	Ca_Quantited:UINT;//负极已叠数量
	Ca_KDQuantited:UINT;//负极空叠隔膜已叠片数
	Ca_EmptyRunKDQuantited:UINT;//负极空跑模式空叠隔膜已叠层数
	Ca_CarryingFalg:BOOL;//负极搬运吸盘有无料标记
	Ca_SegbeltFalg:BOOL;//负极段皮带取模切机械手有无料标记
	Ca_deviationFalg:BOOL;//负极纠偏平台有无料标记
	Ca_DPCarryingFalg:BOOL;//负极叠台搬运吸盘有无料标记
	Ca_DPRequest:BOOL;//负极叠片请求
	//Ca_deviationCCDOK:BOOL;//负极纠偏平台拍照OK
	//Ca_deviationCCDNG:BOOL;//负极纠偏平台拍照NG	
	Ca_deviationCCDDone:BOOL;//负极纠偏平台拍照完成
	Ca_CCDStart:BOOL;//CCD拍照启动
	//Ca_BlueflagingKDSet:UINT;//负极接带空叠隔膜设定片数
	//Ca_YellowmarkKDSet:UINT;//负极色标空叠隔膜设定片数
	Ca_Blueflaging_TF:UINT;//负极蓝胶标记空叠层数		

	Ca_deviationFPOK:BOOL;//负极纠偏平台允许放极片
	Ca_deviationDPOK:BOOL;//负极纠偏平台允许取极片
	Ca_deviationDone:BOOL;//负极纠偏平台纠偏完成
	Ca_CacheBeltDLOK:BOOL;//负极流水线缓存皮带允许取极片
	Ca_CacheBelting:BOOL;//负极流水线缓存皮带取极片中
	Ca_CacheBeltFLOK:BOOL;//负极流水线缓存皮带允许放极片
	Ca_CacheBeltFLing:BOOL;//负极流水线缓存皮带放极片中
	Ca_MainBeltOK:BOOL;//负极流水线主分料皮带允许取极片
	Ca_MainBelting:BOOL;//负极流水线主分料皮带取极片中
	Ca_betlMoveOK:BOOL;//负极搬运升降1在安全位、负极搬运升降2在安全位允许负极流水线线皮带移动
	Ca_AxisCarrying:BOOL;//负极各轴正在运行到初始位中	
	Ca_BeltDone:BOOL;//正极取主分料流水线极片完成
	Ca_BeltSafe:BOOL;//正极取主分料流水线极片安全位
	GetPiceReady:BOOL;//负  极 准备好取分段流水线上的极片
	JumpPiceReady:BOOL;//负  极 放弃取分段流水线上的极片
	bCa_PoleHave:BOOL;//负极取料位无片
	
	Ca_StandbyStep:ARRAY[0..9] OF UINT;//负极备极片程序步
	CarryingSafepos:ARRAY[0..9] OF BOOL;//负极搬动轴在安全位置指示
	Error:ARRAY[0..80] OF BOOL;//报警
		Error_tips	:ARRAY[0..60] OF BOOL;//报警提示
	
	RectifydevStart:BOOL; //纠偏启动
	RectifydevDone:BOOL; //纠偏完成
	//CCD_X1:REAL; //纠偏平台X1的纠偏量
	//CCD_X2:REAL;//纠偏平台X2的纠偏量
	//CCD_Y:REAL;//纠偏平台Y的纠偏量	
	
	DemarcateStart:BOOL; //标定启动	
	DemarcateDone:BOOL; //CCD标定完成
	Demarcateing:BOOL;//CCD标定中
	
	CreateCamStart:BOOL;//负极取片凸轮创建启动
	CreateCamDone:BOOL;//负极取片凸轮创建完成
	
	bCaCCD_TestDo:BOOL;//负极CCD测试开始
	iCaCCD_PhotoCT:INT;//负极拍照取图时间
	iCaCCD_RectifyCT:INT;//负极纠偏时间	
	Ca_CCD_amount :INT;//负极连续NG计数
	Ca_DTqr :BOOL;//负极极片掉片人工确认按钮
	Ca_Rectifydev_CQ :BOOL;//负极纠偏平台除尘
	Ca_Rectifydev_CS :INT;//纠偏计数
	
	Ca_Rectifydev_PB :BOOL;//二次纠偏屏蔽 OFF:屏蔽二次纠偏
	Ca_VacuumErrorNG :BOOL;//负极抛真空NG料标志
	//新增，首层隔膜
	Ca_FirstFoldCnt:INT;//负极首层隔膜已叠次数
	Ca_FirstFoldSet:INT:=1;//负极首层隔膜设定次数
	//20240414WCZ
	RectifyTryStart:BOOL;//CCD重复精度测试启动
	SuckerTestStart:BOOL;//吸盘重复精度测试启动
END_STRUCT
END_TYPE

// ---- P2DUTs/39User2/conDT_Date.TcDUT
TYPE conDT_Date ://叠台叠片
STRUCT
	
	bRecDevBtn:BOOL;//隔膜检测传感器标定按钮
	DT_Blue_TF		  :BOOL;//蓝胶踢废		OFF:屏蔽
	Yellowmark_TF:BOOL;//隔膜色标踢废
	DTIniti_Hbtn:BOOL;//叠台初始化，触摸屏按钮
	DTIniti_Done:BOOL;//叠台初始化完成
	DT_AutoHMI:BOOL;//叠台触摸屏自动
	DT_ManuaHMI:BOOL;//叠台触摸屏手动	
	
	ALLIniti_Hbtn:BOOL;//叠片回原点启动，触摸屏按M钮
	ALLIniti_Done:BOOL;//叠片回原点完成
	CWW:BOOL; //纠偏方向选择
	RecDevEqupos:REAL; //纠偏传感器平衡位置
	RecDevPV:REAL;//纠偏传感器当前值
	RecDevPV1:REAL;//纠偏传感器当前值
	Error:ARRAY[0..100] OF BOOL;//报警
	DT_camError:BOOL;//叠台凸轮报警需初始化
	
	BluGlueNG:ARRAY[0..1] OF BOOL;//表示蓝胶当前电芯或下个电芯NG
	
	CreateCamStart1:BOOL;//叠台压刀凸轮创建启动
	CreateCamDone1:BOOL;//叠台压刀凸轮创建完成
	CreateCamStart2:BOOL;//叠台缓存凸轮创建启动
	CreateCamDone2:BOOL;//叠台缓存凸轮创建完成
	
	Step:ARRAY[0..9] OF UINT;//程序步
	SinStepMode:BOOL;//单步模式
	DP_Mode:BOOL;//叠片完成后，空叠隔膜
	DT_Chesoe:BOOL;//叠负极片选择 
	DT_CellNG_TF	  :BOOL;//对齐度NG梯度踢废 OFF:屏蔽
	
	
	OffloadRequest:BOOL;//叠电芯完成请求下货
	OffloadDone:BOOL;//叠台下货完成
	
	rTension_Start:BOOL;//一键张力启动
	bTenExecute:BOOL;//隔膜张力启动
	bStudyExecute:BOOL;//隔膜张力学习
	PidSwitch:BOOL:=TRUE;//被动放卷开关选择
	fWindDiameter:REAL;//隔膜放卷轴当前卷径
	bTenReady:BOOL;//张力准备好
	bTensionOK:BOOL;//张力OK
	bTenCcw:BOOL;//放卷方向选择
	PTenidSwitch:BOOL;//张力PID开关
	TenAnglePos:REAL;//张力摆杆当前角度	
	TeniGMMoveCount:DINT;//隔膜同步拉伸次数
	
	RectifydevStarte:BOOL;//隔膜纠偏开启HMI
	RectifydevModel:BOOL;//隔膜纠偏屏蔽
	ClearCount:BOOL;//正、负极清零
	
	CDD_OverStart:BOOL;//CCD对奇度检测
	CDD_OverStart_First:BOOL;//CCD对奇度检测压刀间距测量拍照
	OverhandResult:INT;//叠台极片检测有无
	OverhandFirstPice:INT;//叠台极片首层标记
	iOverError:INT;//对齐度检测报警	1：OK，2：NG    实时检测，检测到结果为2就报警

	
	DT_Start           :BOOL;//叠台启动
	
	DT_coumtHight:REAL;//叠片叠台升降已下降高度
	DT_CCD_TwoModel:BOOL;//叠台CCD拍照复检模式
	Door_error :ARRAY[0..80] OF BOOL;//叠台门禁报警
	DT_AllCamOut:BOOL;//叠台一键解耦
	DT_Memory   :INT;//叠台电芯记忆
	DT_amount   :UINT;//已叠电芯数
	DT_amount_clear :BOOL;//电芯数清零
	DT_No      :STRING;//叠台编号
	Machine_No: STRING;//机台编号
	//Cell_Hough    :INT;//(CCD综合评定结果/对齐度)1、对齐度OK，2、对齐度NG
	fWindDiameter_min :REAL;//最小卷径
	Door_Forbidden   :BOOL;//门禁禁用
	Dust_name :INT;//送片皮带毛刷电机
	DiaphragmUnwindingTension :REAL;//隔膜张力
	Manual	:BOOL;//叠台手动
	Put_time :STRING;//投入时间
	DT_Overhang : BOOL;//对齐度屏蔽
	CCD_Overhang_button :BOOL;//叠台电芯确认无极片按钮
	DT_Oerhang_Z :INT;//对齐度结果
	Overhang_TF :BOOL;//对齐度NG踢废信号
	Overhang_Warm:BOOL;//对齐度超限报警
	Overhang_Warm_Reset:BOOL;
	DT_QLqr :BOOL;//叠台已叠片数清零弹窗
	DT_init_OK :BOOL;//叠台工位初始位完成
	YD_JS_L_clear :BOOL;//左压刀计数清零
	YD_JS_R_clear :BOOL;//右压刀计数清零	
	stBnt_Blueflag:BOOL;//蓝胶标记启动
	BlueflagBnt_Warm:BOOL;//是否启动蓝胶标记提示
	
	DT_DayHough:REAL;//对齐度NG数统计白班
	DT_DayHoughAn:REAL;//白班对齐度NG踢废正极片数
	DT_DayHoughCa:REAL;//白班对齐度NG踢废负极片数
	DT_NightHough:REAL;//对齐度NG数统计晚班
	DT_NightHoughAn:REAL;//夜班对齐度NG踢废正极片数
	DT_NightHoughCa:REAL;//夜班对齐度NG踢废负极片数
	DT_DayHough_U:UINT;//对齐度NG数统计白班整数
	DT_NightHough_U:UINT;//对齐度NG数统计晚班整数
	
	DTJD_DayHough:REAL;//白班接带对齐度NG数统计
	DTJD_DayHoughAn:REAL;//白班接带对齐度NG踢废正极片数
	DTJD_DayHoughCa:REAL;//白班接带对齐度NG踢废负极片数
	DTJD_NightHough:REAL;//夜班接带对齐度NG数统计
	DTJD_NightHoughAn:REAL;//夜班接带对齐度NG踢废正极片数
	DTJD_NightHoughCa:REAL;//夜班接带对齐度NG踢废负极片数
	DTJD_DayHough_U:UINT;//白班接带对齐度NG数统计整数
	DTJD_NightHough_U:UINT;//夜班接带对齐度NG数统计整数
	
	DT_GMchange:BOOL;//隔膜更换时间
	DT_OverhangNG:BOOL;//对齐度NG下料时间
	Query:BOOL;//时间查询
	date1:INT;//查询日期
	
	//20231216新增叠台各种状态
	iDTRunStatus:INT;//叠台运行状态：1:自动	2：手动	3：正常电芯空叠隔膜中	4:下料	5：空跑(空叠隔膜)	6:正极踢废		7：负极踢废
	FirstEmpFold:BOOL;//首层空叠隔膜屏蔽

	//20240102新增
	HMI_WinBtn:ARRAY[1..50] OF BOOL;//触摸屏弹窗确认按钮
	HMI_WinOEE_Btn:ARRAY[1..50] OF BOOL;//OEE采集确认按钮
	DiaphragmPartNumberOK    :BOOL;   //隔膜料号OK
	BluePartNumberOK    :BOOL;   //蓝胶料号OK
	PartNumberOff       :BOOL;   //料号功能屏蔽
	Error_tips	:ARRAY[1..30] OF BOOL;//报警提示
	
	fWindLength_M:REAL; //隔膜放卷轴当前米数
	DT_DebugMode           :BOOL;//叠台调试模式料
	DT_Sheetkick     :BOOL;//对齐度单片踢废屏蔽
	DT_YDOpenwindow  :BOOL;//叠台压刀开窗测量屏蔽
	DT_OHclosure		:BOOL;		//对齐度闭环屏蔽		ON是屏蔽
	GMAngleALMsel     :BOOL;		//隔膜卷径报警屏蔽		ON是屏蔽
	
	YD_ferrJSclear :BOOL;//压刀铁氟龙计数清零
	An_sucker1_JSclear      :BOOL;//正极送片搬运吸盘计数清零  
    An_sucker2_JSclear      :BOOL;//正极叠台搬运吸盘计数清零  
    Ca_sucker1_JSclear      :BOOL;//负极送片搬运吸盘计数清零  
    Ca_sucker2_JSclear      :BOOL;//负极叠台搬运吸盘计数清零  
    Ca_sucker3_JSclear      :BOOL;//负极流水线搬运吸盘计数清零  	
END_STRUCT
END_TYPE

// ---- P2DUTs/39User2/conDT_RunStatus.TcDUT
TYPE conDT_RunStatus :
STRUCT
	DT_AutoRuning: BOOL;//叠台自动运行中--无跳片
	DT_ReadyTemp: BOOL;//叠台输出取片准备好信号
	DT_ReadyAllow: BOOL;//模切调度让叠台容许取片信号
	ReadyAllow2:BOOL;//模切调度让叠台容许取片信号
	//叠台当前状态	
	iDTRunStatus:INT;//叠台当前状态
	
	//20240504 CF
	bSyncReady:BOOL;//同步准备好
	bJumpSync:BOOL;//放弃同步
	bSyncStart:BOOL;//开始同步
END_STRUCT
END_TYPE

// ---- P2DUTs/39User2/conStickGlue_date.TcDUT
TYPE conStickGlue_date :
STRUCT
	
	StickMark_L1:BOOL;//左短边1贴胶完成
	StickMark_L2:BOOL;//左短边2贴胶完成
	StickMark_R1:BOOL;//右短边1贴胶完成
	StickMark_R2:BOOL;//右短边2贴胶完成
	StickMark1_L:BOOL;//非极耳侧贴胶完成---------
	StickMark1_L2:BOOL;//极耳侧贴胶完成---------
	StickPermit:BOOL;//贴胶允许
	StickFinish:BOOL;//贴胶完成
	Sticking_L:BOOL;//左短边贴胶
	Sticking_R:BOOL;//右短边贴胶
	Sticking_Lg:BOOL;//非极耳侧长边贴胶--------
	Sticking_Lg2:BOOL;//极耳侧长边贴胶--------
	
	
	//Stickersettings:word_bool;//贴胶设置需要贴的胶道数
	Stickersetting:ARRAY[0..9] OF BOOL;//贴胶设置需要贴的胶道数
	
	//StickerDoneNo:word_bool;//已贴胶的道数
	StickerDoneNo:ARRAY[0..9] OF BOOL;//已贴胶的道数
		
	Stickerragree:BOOL;//贴胶允许尾卷下电芯
	StickerFlag:BOOL;//贴胶夹爪有无电芯标志
	StickerDone:BOOL;//贴胶完成
	StickerOffloading:BOOL;//贴胶下电芯请求
	StickerOffloadingDone:BOOL;//贴胶下电芯完成	
	StickerStandbyDone:BOOL;//贴胶备胶完成
	StickerStandbyCode:BOOL;//备二维码胶请求
	StickerStandbyBule:BOOL;//备蓝胶请求
	TJIniti_Done:BOOL;//贴胶初始化完成
	TJIniti_Hbtn:BOOL;//贴胶初始化，触摸屏按鋕
	
	SinStepMode:BOOL;//单步模式
	
	ScanStarte:BOOL;//扫码启动
	ScanOK:BOOL;//扫码OK
	ScanNG:BOOL;//扫码NG
	Scan_gross :INT;//1、OK 2、NG
	ScanMode:BOOL;//扫码模式，是否屏蔽
	ScanStatus:ARRAY[0..2] OF BOOL;//记录扫码的状芯
	
	Error:ARRAY[0..29] OF BOOL;//报警
	
	StickerStart_HMI:BOOL;//尾卷贴胶启动
	
	AxisConditionEN:BOOL;//TRUE:电机运动条件屏蔽
	TJ_Memory   :INT;//贴胶电芯记忆
	WhirlingSafe :BOOL;//贴胶旋转安全条件
	strCode :STRING;//扫码码条
	Scan_IP :T_IPv4Addr;
	bTcpOpen :BOOL;//扫码Tcp 连接
	Scan_Men :ARRAY[1..4] OF Scan_TJ;//贴胶扫码记忆
	Scan_TS   :BOOL; //扫码提示
	Scan_CT :BOOL;//扫码数据传递
	
	Stick_Judge:BOOL;//贴胶软限位判断
	
END_STRUCT
END_TYPE

// ---- P2DUTs/39User2/conTailCurl_date.TcDUT
TYPE conTailCurl_date ://尾卷数据包
STRUCT
	HotCut:BOOL;//热切丝启动	
	TailCurlStart:BOOL;//尾卷启动
	TailCurlDone:BOOL;//尾卷完成	
	
	TailCultOffloading:BOOL;//尾卷下电芯请求
	TailCultOffloadingDone:BOOL;//尾卷下电芯完成

	WZIniti_Done:BOOL;//尾卷初始化完成
	WZIniti_Hbtn:BOOL;//尾卷初始化，触摸屏按钮
	
	CreateCamStart:BOOL;//尾卷凸轮创建启动
	CreateCamDone:BOOL;//尾卷凸轮创建完成
	
	TailCurlStep:ARRAY[0..9] OF UINT;//尾卷贴胶程序步
	
	SinStepMode:BOOL;//单步模式
	
	Error:ARRAY[0..29] OF BOOL;//报警
	
	AxisConditionEN:BOOL;//TRUE:电机运动条件屏蔽
	
	WJ_AllCamOut:BOOL;//尾卷一键解耦
	WJ_Memory   :INT;//尾卷电芯记忆
	Manual	:BOOL;//尾卷手动
	
	b_WJqr :BOOL;//选择是否不尾卷,false:尾卷，true：不尾卷
	
	WJ_TIME:REAL;//尾卷计时
	HotClear:BOOL;//热切切断计数清零	
	TailCurlSEPTALineSavePos:ARRAY[1..2] OF LREAL;//夹膜平移记录位置
END_STRUCT
END_TYPE

// ---- P2DUTs/39User2/parDT_date.TcDUT
TYPE parDT_date :// 关于叠台设定断电保持的参数
STRUCT
	rRecDev:REAL;//隔膜检测传感器标定值显示，触摸屏只显示不输入
	rRecDevScope:REAL:=1;//隔膜检测传感器标定范围，超过该值判断隔膜打皱
	An_Quantity:UINT;//正极设定极片数		
	An_KDQuantity:UINT;//正极空叠极片设定
	Ca_Quantity:UINT;//负极设定极片数
	Ca_KDQuantity:UINT;//负极空叠极片设定
	Ca_betlCount:WORD;//负极极片级存流水线记录极片数
	
	Ca_MQ_Slice	:ARRAY[0..9] OF ST_BeltData;//负极模切极片数据  7:送片搬运数据 8:纠偏台数据 9:叠片搬运数据
	An_MQ_Slice	:ARRAY[0..2] OF ST_BeltData;//正极模切极片数据  0:正极送片搬运数据  1:正极纠偏台数据  2:正极叠片搬运数据
	
	CaMQ_MES :ST_BeltData;//负极MES交互数据
	AnMQ_MES :ST_BeltData;//正极MES交互数据
	
	
	Ca_Thickness:REAL;//负极片厚度
	An_Thickness:REAL;//正极片厚度
	SEPTA_Thickness:REAL;//隔膜厚度
	Pole_ThicknessCom:REAL;//极片厚度补偿系数

	
	Distance:REAL;//蓝胶检测到压刀外边的距离
	BluWidth:REAL; //蓝胶宽度
	Width:REAL:=189; //压刀外边宽
	
	SinglePosTime:REAL;//单片时间，主轴速度
	
	
	TensionTable:ARRAY[0..105,1..2] OF REAL;//张力摆杆的学习数据
	fStudyDiameter:REAL;//学习时隔膜的卷径
	fDancerMinPos:REAL; //摆杆最小角度
	fDancerMaxPos:REAL;//摆杆最大角度
	fDanceBlancePos:REAL; //摆杆平衡位置
	PidSwitch:REAL; //单次叠膜隔宽度
	
	//隔膜纠偏
	iRectifyAnPos:REAL:=50;//正极位纠偏范围
	iRectifyCaPos:REAL:=50;//负极位纠偏范围
   	 iRectifyMode     :INT;    //隔膜纠偏模式选择

	RecDevValueSet:REAL;//纠偏偏差值设置
	RecDevSpeedCoe:REAL; //纠偏速度系数

	fRectifyMaxValue:REAL;//从轴纠偏行程上限
	fRectifyMinValue:REAL;//从轴纠偏行程下降
	fRectifyBalanceValue:REAL;//纠偏平衡位置
    fRectifyfTolerance:REAL;//纠偏平衡位置
	fRectifyGMLengthSet :REAL;//纠偏隔膜长度标定
    fRectifyTimeAdjust           :REAL;  //纠偏时间标定
    DP_fRectifyTimeAdjust        :REAL;  //叠片纠偏时间标定
	
	BeltPoistSet:REAL;//负极皮带相对位置
	BeltPoistTime:REAL;//负极皮带时间

    fDiameterWarn:REAL;//隔膜放卷卷径临界设置（警告）
    fDiameterAlarm:REAL;//隔膜放卷卷径临界设置（报警）

	DT_Overhang_SUM :UINT:=30;//负极已叠片数踢对齐度数量
	BH_Thickness  :REAL;//变化厚度
	Overhang_CSJS :UDINT;//对齐度检测超时计数
	YD_JS_L         :UDINT;//左压刀计数
	YD_YJ_L		  	:UDINT:=1000000;//左压刀预警值
	YD_SM_L		  	:UDINT:=1000000;//左压刀寿命
	YD_JS_R         :UDINT;//右压刀计数
	YD_YJ_R		  	:UDINT:=1000000;//左压刀寿命
	YD_SM_R		    :UDINT:=1000000;//右压刀预警值
	YDBarCode_L		:STRING(49);//左压刀压刀条码
	YDBarCode_R		:STRING(49);//右压刀压刀条码
	YDCuterTime_L	:STRING(49);//左压刀换刀时间
	YDCuterTime_R	:STRING(49);//右压刀换刀时间
	An_Rectifydev_JS :UDINT;//正极纠偏平台NG计数
	Ca_Rectifydev_JS :UDINT;//负极纠偏平台NG计数
	An_Rectifydev_Btn :BOOL;//正极纠偏平台NG计数清零
	Ca_Rectifydev_Btn :BOOL;//负极纠偏平台NG计数清零
	An_Rectifydev_NGSet :UDINT:=10;//正极纠偏平台NG片数设定
	Ca_Rectifydev_NGSet :UDINT:=10;//负极纠偏平台NG片数设定
	
	An_stuff_No				 :STRING;//正极极卷号
	Ca_stuff_No				 :STRING;//负极极卷号
	Diaphragm_No			 :STRING;//隔膜批次
	QR_code_No				 :STRING;//二维码批次
	Glue_No					 :STRING;//收尾胶批次
	iTargetTorqueBLXS	:INT:=10;		//尾卷时扭矩值比例系数
	iTargetTorqueHMI	: INT:=-80;	//扭矩值HMI变量
	
	fVelocity_of_QDX   :REAL:=5; //	夹电芯取电芯速度
	fVelocity_of_LM   :REAL:=5; //	夹电芯拉膜速度
	
	stSetLenght:REAL;//蓝胶接带点到叠台的距离
	DtCountSet:ARRAY[1..10] OF INT :=[10(10)];//叠台备用计数设定 1:叠台真空关闭层数设定
	DtCount:ARRAY[1..10] OF INT;//叠台备用计数 
	CleanTimeHMIHour:INT;//清洁时间Hour
	CleanTimeHMIMin:INT;//情节时间Min	

	//叠台COE寻址修改参数
	EtherCatNetID :STRING; //EtherCAT支路ID
	EtherCatAddr :ARRAY[1..6] OF INT ;    //EtherCAT支路里驱动器ID
	wSaveCoeCode  :DWORD:=16#65766173;    //电机参数保存
	SEPTATLine_fSmoothValue   :ARRAY[1..2] OF REAL;    //隔膜平移写入参数值
	SEPTATLine_bWriteCoeValue  :ARRAY[1..2] OF BOOL;    //隔膜平移写入执行	
	SEPTATLine_SavePara  :ARRAY[1..2] OF BOOL;   //隔膜平移参数保存	
	SEPTATCache_fSmoothValue   :ARRAY[1..2] OF REAL;    //隔膜缓存写入参数值
	SEPTATCache_bWriteCoeValue  :ARRAY[1..2] OF BOOL;    //隔膜缓存写入执行	
	SEPTATCache_SavePara  :ARRAY[1..2] OF BOOL;   //隔膜缓存参数保存	
	AnCarryingLine_fSmoothValue   :ARRAY[1..2] OF REAL;    //正极送片搬运平移写入参数值
	AnCarryingLine_bWriteCoeValue  :ARRAY[1..2] OF BOOL;    //正极送片搬运平移写入执行	
	AnCarryingLine_SavePara  :ARRAY[1..2] OF BOOL;   //正极送片搬运平移参数保存
	AnDTCarryingLine_fSmoothValue   :ARRAY[1..2] OF REAL;    //正极叠片搬运平移写入参数值
	AnDTCarryingLine_bWriteCoeValue  :ARRAY[1..2] OF BOOL;    //正极叠片搬运平移写入执行	
	AnDTCarryingLine_SavePara  :ARRAY[1..2] OF BOOL;   //正极叠片搬运平移参数保存
	CaCarryingLine2_fSmoothValue   :ARRAY[1..2] OF REAL;    //负极送片搬运平移写入参数值
	CaCarryingLine2_bWriteCoeValue  :ARRAY[1..2] OF BOOL;    //负极送片搬运平移写入执行	
	CaCarryingLine2_SavePara  :ARRAY[1..2] OF BOOL;   //负极送片搬运平移参数保存
	CaDTCarryingLine_fSmoothValue   :ARRAY[1..2] OF REAL;    //负极叠片搬运平移写入参数值
	CaDTCarryingLine_bWriteCoeValue  :ARRAY[1..2] OF BOOL;    //负极叠片搬运平移写入执行	
	CaDTCarryingLine_SavePara  :ARRAY[1..2] OF BOOL;   //负极叠片搬运平移参数保存
	
	GMlength_set:REAL;//隔膜总长度
	GMlength_act:REAL;//隔膜当前长度
	GMlength_manual:REAL;//手动拉膜长度
	GMlength_manual2:REAL;//手动拉膜长度
	GMlength_buttonl:BOOL;//手动拉膜确定按钮
	
	Ca_BlueflagingKDSet:UINT:=13;//负极接带空叠隔膜设定片数
	Ca_YellowmarkKDSet:UINT:=20;//负极色标空叠隔膜设定片数
	
	fInsideDiameter:REAL:=88; //内直径
	fTen_K:REAL;//张力K值
	fTen_B:REAL;//张力B值
	fTenset:REAL;//张力设定值
	bRepair:BOOL;//叠台维修
	An_Rectifydev_DayNG:UDINT;//正极纠偏平台白班NG计数
	Ca_Rectifydev_DayNG:UDINT;//负纠偏平台白班NG计数
    An_Rectifydev_NightNG :UDINT;//正极极纠偏平台晚班NG计数	
	Ca_Rectifydev_NightNG :UDINT;//负极纠偏平台晚班NG计数	
	fAlmpos:REAL; //隔膜放卷报警值，度/毫米
	//20240414WCZ
	An_Demarcate_X:REAL;//纠偏重复精度测试设定纠偏值X
	An_Demarcate_X2:REAL;//纠偏重复精度测试设定纠偏值X
	An_Demarcate_Y:REAL;//纠偏重复精度测试设定纠偏值Y
	An_Demarcate_R:REAL;//纠偏重复精度测试设定纠偏值R
	An_CCDNo:INT;//纠偏重复精度测试次数
	An_CCDCount:INT;//吸盘重复精度测试次数
	
	Ca_Demarcate_X:REAL;//纠偏重复精度测试设定纠偏值X
	Ca_Demarcate_X2:REAL;//纠偏重复精度测试设定纠偏值X	
	Ca_Demarcate_Y:REAL;//纠偏重复精度测试设定纠偏值Y
	Ca_Demarcate_R:REAL;//纠偏重复精度测试设定纠偏值R	
	Ca_CCDNo:INT;//纠偏重复精度测试次数
	Ca_CCDCount:INT;//吸盘重复精度测试次数
	
	YD_ferrJS         :UDINT;//左压刀铁氟龙计数
    YD_ferrset         :UDINT:=1000000;//左压刀铁氟龙设定值
	An_sucker1_JS      :UDINT;//正极送片搬运吸盘计数
	An_sucker1Set      :UDINT:=1000000;//正极送片搬运吸盘设定值
	An_sucker2_JS      :UDINT;//正极叠台搬运吸盘计数
	An_sucker2Set      :UDINT:=1000000;//正极叠台搬运吸盘设定值
	Ca_sucker1_JS      :UDINT;//负极送片搬运吸盘计数
	Ca_sucker1Set      :UDINT:=1000000;//负极送片搬运吸盘设定值
	Ca_sucker2_JS      :UDINT;//负极叠台搬运吸盘计数  
	Ca_sucker2Set      :UDINT:=1000000;//负极叠台搬运吸盘设定值
    Ca_sucker3_JS      :UDINT;//负极流水线搬运吸盘计数  
    Ca_sucker3Set      :UDINT:=1000000;//负极流水线搬运吸盘设定值
	
	GMAngleALM:REAL:=0.81;//隔膜剩余角度报警值
END_STRUCT
END_TYPE

// ---- P2DUTs/39User2/parMechanical.TcDUT
TYPE parMechanical :// 关于叠台设定断电保持的参数
STRUCT

   //隔膜机械参数
    fGMRollDiameter     :  REAL:=24;    //隔膜辊直径 

   	y_C1          : REAL:=22.25;     //C1辊中心Y坐标

   	x_D1          : REAL:=-112.5; //左压针外边X坐标
   	x_D2          : REAL:=112.5;//右压针外边X坐标

    y_B1         : REAL:=102.25;//下上辊Y坐标
   	y_A5         : REAL:=368.25;//上辊中心Y坐标


   //尾卷机械参数
	fCellWidth     :REAL :=  81.92 ;   //电芯宽
	fCellThick      :REAL :=  23.4;     //电芯厚度
	fCellRadii       :REAL :=   2 ;       //电芯厚度




END_STRUCT
END_TYPE

// ---- P2DUTs/39User2/parTailCurl_date.TcDUT
TYPE parTailCurl_date :
STRUCT
	HotTime:REAL;//热切加热时间
	SumNo:REAL:=1;//尾卷总圈数
	SynNo:REAL;//尾卷同步圈数
	CoeSpeed:REAL;//尾卷主轴速度系数
	Xlength:REAL;//夹膜平移夹板到卷针边距离
	WJ_PoistCamOut:REAL;//尾卷夹膜平移凸轮解耦位置
	Sticker_Model: BOOL;//贴胶MARK与定长切换
	Hotcount:UDINT;///热切切断计数
	Hotlifetime:UDINT;///热切切断寿命
END_STRUCT
END_TYPE

// ---- P2DUTs/39User2/Scan_TJ.TcDUT
TYPE Scan_TJ :
STRUCT
Scan_gross :INT;//扫码，1、OK，2、NG
TJ_Code    :STRING;	//码条

END_STRUCT
END_TYPE

// ---- P2DUTs/39User2/ST_Timedata.TcDUT
TYPE ST_Timedata :
STRUCT
	
	RunTime:ARRAY[0..25] OF UINT;//运行时间
    WaitTime:ARRAY[0..25] OF UINT;//待机时间
    AlmTime:ARRAY[0..25] OF UINT;//报警时间 	
    OverhangNGTime:ARRAY[0..25] OF UINT;//t剔对齐度时间 	
    GMchangeTime:ARRAY[0..25] OF UINT;//隔膜更换时间 	
	
END_STRUCT
END_TYPE

// ---- P2DUTs/39User2/ST_Torque.TcDUT
TYPE ST_Torque :
STRUCT
	
	An_CarryingTorSet:INT;//正极搬运1移位报警力矩设定
	An_DTCarryingTorSet:INT;//正极叠台搬运报警力矩值设定
	Ca_Carrying1TorSet:INT;//负极搬运1平移报警力矩设定
	Ca_Carrying2TorSet:INT;//负极搬运2平移报警力矩设定
	Ca_DTCarryingTorSet:INT;//负极叠台搬运平移报警力矩设定
	TailCurlTorSet:INT;//尾卷夹电芯平移报警力矩设定
	TailCurlWhirlTorSet:INT;//尾卷夹电芯旋转报警力矩设定
	TailCurlSEPTATorSet:INT;//夹膜平移报警力矩设定
	//TailCurlRetTorSet:INT;//尾卷夹电芯伸缩力矩设定
	
	An_CarryingTor:INT;//正极搬运1移位实时力矩
	An_DTCarryingTor:INT;//正极叠台搬运实时力矩
	Ca_Carrying1Tor:INT;//负极搬运1平移实时力矩
	Ca_Carrying2Tor:INT;//负极搬运2平移实时力矩
	Ca_DTCarryingTor:INT;//负极叠台搬运平移实时力矩
	TailCurlTor:INT;//尾卷夹电芯平移实时力矩
	TailCurlWhirlTor:INT;//尾卷夹电芯旋转实时力矩
	TailCurlSEPTATor:INT;//夹膜平移实时力矩
	//TailCurlRetTor:INT;//尾卷夹电芯伸缩实时力矩
	
	An_CarryingTorAlarm:BOOL;//正极搬运1移位力矩超限报警
	An_DTCarryingTorAlarm:BOOL;//正极叠台搬运力矩超限报警
	Ca_Carrying1TorAlarm:BOOL;//负极搬运1平移力矩超限报警
	Ca_Carrying2TorAlarm:BOOL;//负极搬运2平移力矩超限报警
	Ca_DTCarryingTorAlarm:BOOL;//负极叠台搬运平移力矩超限报警
	TailCurlTorAlarm:BOOL;//尾卷夹电芯平移力矩超限报警
	TailCurlWhirlTorAlarm:BOOL;//尾卷夹电芯旋转力矩超限报警
	TailCurlSEPTATorAlarm:BOOL;//夹膜平移力矩超限报警
	//TailCurlRetTorAlarm:BOOL;//尾卷夹电芯伸缩力矩超限报警
END_STRUCT
END_TYPE

// ---- P2DUTs/39User2/ST_UserControl.TcDUT
TYPE ST_UserControl :
STRUCT
	DT_iMode:UINT;//叠台控制模式  1自动  2停止    3手动 	4急停
	WJ_iMode:UINT;//尾卷控制模式  1自动  2停止    3手动 	4急停
	TJ_iMode:UINT;//帖胶控制模式  1自动  2停止    3手动 	4急停
	
	Funselection:UINT;//功能选择    1、空跑  
	Step:ARRAY[0..9] OF UINT;//程序步
	//ALLIniti_Done:BOOL;//始化完成
	P2Init:BOOL;//上电初始化
	P2InitDone:BOOL;//上电初始化完成
	EmptyRunMode:BOOL;//空跑模式
	DT_ModelChees:BOOL;//叠台是否启用选择，0：启用  1：屏蔽
	
	CCD_ChosesHMI:BOOL;//CCD屏蔽
	
	
	//当前产量
	//当前节拍
	//当前速度
	
	
	
	//Ca_StandbyStep:ARRAY[0..9] OF UINT;//负极备极片程序步
	//An_StandbyStep:ARRAY[0..9] OF UINT;//正极备极片程序步
	//TailCurlStep:ARRAY[0..9] OF UINT;//尾卷贴胶程序步
	
	//DTIniti_Hbtn:BOOL;//叠台初始化，触摸屏按钮
	//WZIniti_Hbtn:BOOL;//尾卷初始化，触摸屏按钮
	//TJIniti_Hbtn:BOOL;//贴胶初始化，触摸屏按鋕
	//ALLIniti_Hbtn:BOOL;//1号叠片初始化，触摸屏按M钮

	//DTIniti_Done:BOOL;//叠台初始化完成
	//WZIniti_Done:BOOL;//尾卷初始化完成
	//TJIniti_Done:BOOL;//贴胶初始化完成
	

	
	
	//DP_Done:BOOL;//叠台叠片完成
	
	//TailCultOffloading:BOOL;//尾卷下电芯请求
	//TailCultOffloadingDone:BOOL;//尾卷下电芯完成	
	(*
	Stickerragree:BOOL;//贴胶允许尾卷下电芯
	StickerFlag:BOOL;//贴胶夹爪有无电芯标志
	StickerDone:BOOL;//贴胶完成
	StickerOffloading:BOOL;//贴胶下电芯请求
	StickerOffloadingDone:BOOL;//贴胶下电芯完成	
	
	StickerStandbyDone:BOOL;//贴胶备胶完成
	
	StickerStandbyCode:BOOL;//备二维码胶请求
	StickerStandbyBule:BOOL;//备蓝胶请求
	*)

	
	
	
	//HotCut:BOOL;//热切丝启动
	
	//TailCurlStart:BOOL;//尾卷启动
	//TailCurlDone:BOOL;//尾卷完成
	(*
	An_Quantited:UINT;//正极已叠数量
	An_CarryingFalg:BOOL;//正极搬运吸盘有无料标记
	An_QuLiaoOK:BOOL;//正极取流水线极片允许
	An_deviationFalg:BOOL;//正极纠偏平台有无料标记
	An_DPCarryingFalg:BOOL;//正极叠台搬运 吸盘有无料标记
	An_DPRequest:BOOL;//正极叠片请求
	An_deviationCCDOK:BOOL;//正极纠偏平台拍照OK
	An_deviationCCDNG:BOOL;//正极纠偏平台拍照NG
	An_deviationFPOK:BOOL;//正极纠偏平台允许放极片
	An_deviationDPOK:BOOL;//正极纠偏平台允许取极片
	An_deviationDone:BOOL;//正极纠偏平台纠偏完成
	An_MainBeltOK:BOOL;//正极流水线主分料皮带允许取极片
	An_MainBelting:BOOL;//正极流水线主分料皮带取极片中
	AN_AxisCarrying:BOOL;//正极各轴正在运行到初始位中
	*)
	(*
	Ca_Quantited:UINT;//负极已叠数量
	Ca_CarryingFalg:BOOL;//负极搬运吸盘有无料标记
	Ca_SegbeltFalg:BOOL;//负极段皮带取模切机械手有无料标记
	Ca_deviationFalg:BOOL;//负极纠偏平台有无料标记
	Ca_DPCarryingFalg:BOOL;//负极叠台搬运吸盘有无料标记
	Ca_DPRequest:BOOL;//负极叠片请求
	Ca_deviationCCDOK:BOOL;//负极纠偏平台拍照OK
	Ca_deviationCCDNG:BOOL;//负极纠偏平台拍照NG	
	Ca_deviationFPOK:BOOL;//负极纠偏平台允许放极片
	Ca_deviationDPOK:BOOL;//负极纠偏平台允许取极片
	Ca_deviationDone:BOOL;//负极纠偏平台纠偏完成
	Ca_CacheBeltDLOK:BOOL;//负极流水线缓存皮带允许取极片
	Ca_CacheBeltFLOK:BOOL;//负极流水线缓存皮带允许放极片
	Ca_MainBeltOK:BOOL;//负极流水线主分料皮带允许取极片
	Ca_MainBelting:BOOL;//负极流水线主分料皮带取极片中
	Ca_betlMoveOK:BOOL;//负极搬运升降1在安全位、负极搬运升降2在安全位允许负极流水线线皮带移动
	Ca_AxisCarrying:BOOL;//负极各轴正在运行到初始位中
	
*)

	
END_STRUCT
END_TYPE

// ---- P2DUTs/指纹/ST_FingerprintKey.TcDUT
TYPE ST_FingerprintKey :
STRUCT
	MachineId		: 	STRING(49);//指纹器编号	
	UserId			:	STRING(49);//用户名	
	UserClassLevel	: 	STRING(49);//用户权限	
	Fid				: 	STRING(49);//本地文件id	
	MatchScore		:	STRING(49);//指纹匹配评分	
	Result			: 	STRING(49);//匹配结果	
	FileName		: 	STRING(49);//本地文件路径	
END_STRUCT
END_TYPE

// ---- P3UDTs/MES/DTM_Mes1.TcDUT
TYPE DTM_Mes1 :
STRUCT
	uOther		:ARRAY[0..19] OF UINT;	//信号交互		
	bFuncEN     :ARRAY[0..10] OF BOOL; //功能开关状态
END_STRUCT
END_TYPE

// ---- P3UDTs/MES/Mes1.TcDUT
TYPE Mes1 :
STRUCT
	rExcelRate	:ARRAY[0..119] OF REAL;	//优报表real
	uOther		:ARRAY[0..19] OF UINT;	//信号交互
	bFuncEN      :ARRAY[0..50] OF BOOL;  //功能开关状态
	Error       :ARRAY[0..50] OF BOOL;  //功能开关状态报警
END_STRUCT
END_TYPE

// ---- P3UDTs/MES/Mes2.TcDUT
TYPE Mes2 :
STRUCT
	Serialnumber	:INT;//片序号
	Polarity	:INT;//极性 1负极 2正极
	Platenumber	:   STRING(49) ;//  模切极片编号
	AnlapTen	:REAL ;// 正极放卷张力每一片
	CalapTen	:REAL ;// 负极放卷张力每一片
	GMlapTen	:REAL ;// 隔膜放卷张力每一片
	GMlapRectify	:REAL ;// 隔膜放卷纠偏每一片
END_STRUCT
END_TYPE

// ---- P3UDTs/MES/MTD_Mes1.TcDUT
TYPE MTD_Mes1 :
STRUCT
	rExcelRate	:ARRAY[0..99] OF REAL;	//优报表real
	uOther		:ARRAY[0..19] OF DINT;	//信号交互
	bFuncEN     :ARRAY[0..20] OF BOOL; //功能开关状态
END_STRUCT
END_TYPE

// ---- P3UDTs/Output_statistic/Statistics.TcDUT
TYPE Statistics :
STRUCT
	FirstCheck	 :UINT;//首检NG
	His_FirstCheck:UINT;//昨天首检NG
	Hough 		 :UINT;//对齐度NG
	His_Hough    :UINT;//昨天对齐度NG
	JDHough 		 :UINT;//接带对齐度NG
	JDHis_Hough    :UINT;//昨天接带对齐度NG	
	ScanCode	 :UINT;//扫码NG
	ShortTest 	 :UINT;//短路测试NG
	Weight 		 :UINT;//称重NG
	Thickness 	 :UINT;//测厚NG
	MES          :UINT;//MES的NG
	Hough_DT  :ARRAY[1..3] OF UINT;//每个叠台对齐度NG数量
	His_HoughAn  :ARRAY[1..3] OF UINT;//每个叠台对齐度NG正极片数
	His_HoughCa  :ARRAY[1..3] OF UINT;//每个叠台对齐度NG负极片数
END_STRUCT
END_TYPE

// ---- P3UDTs/Output_statistic/ST_Timedata_1.TcDUT
TYPE ST_Timedata_1 :
STRUCT
	
	RunTime:ARRAY[0..25] OF UINT;//运行时间
    WaitTime:ARRAY[0..25] OF UINT;//待机时间
    AlmTime:ARRAY[0..25] OF UINT;//报警时间 	
    XLWaitTime:ARRAY[0..25] OF UINT;//下料等待时间  	

	
END_STRUCT
END_TYPE

// ---- P3UDTs/P3_AxisCO_Ntrol/ST_AxisCmdV2.TcDUT
TYPE ST_AxisCmdV2 :  //轴运动控制相关
STRUCT

   bDynamitcsParSel      :INT:=1;  // 1:NC          2:UserDefine


	bEnable			        :BOOL;				    (*使能*)
	fOverride			    :REAL:=100;			(*MC_power中实际倍率的设定，默认值为100*)
	bEnableFw		        :BOOL:=TRUE;		 (*正向使能*)
	bEnableBw		    :BOOL:=TRUE;	 	(*负向使能*)

	bJog_Fw			    :BOOL;			     	(*正向点动*)
	bJog_Bw			    :BOOL;			    	(*反向点动*)

	bMoveAbs	 	        :BOOL;				    (*运行绝对位置*)
	fPositon_of_Abs	 	:REAL;					(*绝对位置位移*)

	bMoveRel		        :BOOL;				   (*运行当对位置*)
	fPosition_of_Rel	    :REAL;				   (*相对位置位移*)

	bMoveModulo		 :BOOL;				     (*运行模长位置*)
	fPositon_of_Mod	  :REAL;					  (*模长位置位移*)

	bMoveVelo		    :BOOL;				       (*向一个方向持续运行，方向由前面的正向点动或者反向点动设置*)
	bMoveVeloDir	:MC_Direction := MC_Positive_Direction ;	(*速度运动的方向,MC_Negative_Direction*)

	bHome			       :BOOL;						(*启动回参*)

	bSetPos			       :BOOL;						 (*设置轴当前的位置为一个绝对位置*)
    fSetPos				   :REAL:=0;					(*setpos功能块将轴当前的位置设置为这个变量*)

	iGoSetPos              :INT;                     //GO离散点位_INT
    arrbGoSetPos      :ARRAY[0..50]        OF BOOL;  //GO离散点位_布尔数组
	iRealPoint              :INT;                     //离散点位指示_INIT
    arrbRealPoint        :ARRAY[0..50]        OF BOOL;  //离散点位指示_布尔数组

	bHalt			            :BOOL;				(*暂停*)
	bStop			        :BOOL;				(*停止*)
	bGearOut			    :BOOL;				(*解耦*)
	bReset			        :BOOL;				(*复位*)

	hmiJog_Fw			    :BOOL;				//正向点动_BOOL
	hmibJog_Bw		     :BOOL;				//反向点动_BOOL	
	hmiGoSetPos          :INT;              //GO离散点位_INT


//条件
     Home_Condition       :BOOL;//回原点条件
     JogP_Condition       :BOOL;//点动正转条件
     JogN_Condition       :BOOL;//点动反转条件
     GoPoint_Condition    :ARRAY[0..50] OF BOOL;//HMI点动定位条件








END_STRUCT
END_TYPE

// ---- P3UDTs/P3_AxisCO_Ntrol/ST_AxisCtrlV2.TcDUT
TYPE ST_AxisCtrlV2 :
STRUCT
    Io                        :ST_AxisIo;  (*轴IO信号*)
    Status                  :ST_AxisStatus;  
    Cmd                    :ST_AxisCmdV2;  
END_STRUCT
END_TYPE

// ---- P3UDTs/P3_AxisCO_Ntrol/ST_Axis_ParV2.TcDUT
TYPE ST_Axis_ParV2 ://轴参数
STRUCT

	fVelocity_of_Abs	 :REAL:=5;				
	fVelocity_of_Mod	 :REAL:=5;				
	fVelocity_of_Rel	 :REAL:=5;				
	fVelocity_of_Velo	 :REAL:=5;				
	fVelocity_of_Jog	 :REAL:=10;			
	fInchingDistance	 :REAL:=5;				

	arrTargetPoint: ARRAY [0..50] OF REAL;
	//fMaxVelocity:        REAL:=0;	
    fTagatTime                                 :REAL:=0.5;//S
    fConVelPercentage                      :REAL:=0.8;//S
    fMaxAccDec                              :LREAL:=40000;//最大加速度
    fMaxVel                                   :LREAL:=2000;//最大速度

	fHomePosition                     :REAL:=10 ;	                          
	fHomeFastSpeed                  :REAL:=20 ;	 
	fHomeSlowSpeed                 :REAL:=10;	 
    HomeLimitDis                       :REAL:=5;	 

END_STRUCT
END_TYPE

// ---- P3UDTs/P3_IO/ST_P3Button.TcDUT
TYPE ST_P3Button :
STRUCT
P3_ColdWarning_Buzzer	:BOOL;	//冷压上料搬运电机运行蜂鸣器	
P3_ColdWarning_Lamp     :BOOL;  //冷压上料搬运电机运行警示灯
NG_button_1				:BOOL;//NG按钮1
NG_button_2				:BOOL;//NG按钮2
LateStop				:BOOL;//尾段急停
IDStickBtn:BOOL;//二维码备胶按钮
IDCutbtn:BOOL;//二维码切胶按钮
IDGluebtn:BOOL;//二维码拉胶按钮
P3_Startbtn:BOOL;//热压，启动按钮
P3_Resetebtn:BOOL;//热压台，复位按钮
P3_Stopbtn:BOOL;//热压台，停止按钮
P3_Autobtn:BOOL;//热压台，手自动按钮
END_STRUCT
END_TYPE

// ---- P3UDTs/P3_IO/ST_P3Senser.TcDUT
TYPE ST_P3Senser :
STRUCT
P3_PoleMotor1_JogP      :BOOL;//对齐度NG排杆电机正转
P3_PoleMotor1_JogN      :BOOL;//对齐度NG排杆电机反转
P3_PoleMotor1_Reach     :BOOL;//对齐度NG料盒到位感应
P3_PoleMotor1_Height    :BOOL;//对齐度NG料盒高度感应
P3_PoleMotor1_P_OT      :BOOL;//对齐度NG料盒顶升电机上限
P3_PoleMotor1_N_OT      :BOOL;//对齐度NG料盒顶升电机下限
P3_PoleMotor1_bHave		:BOOL;//对齐度NG料盒有料感应
P3_PoleMotor2_JogP      :BOOL;//短路NG排杆电机正转
P3_PoleMotor2_JogN      :BOOL;//短路NG排杆电机反转
P3_PoleMotor2_Reach     :BOOL;//短路NG料盒到位感应
P3_PoleMotor2_Height    :BOOL;//短路NG料盒高度感应
P3_PoleMotor2_P_OT      :BOOL;//短路NG料盒顶升电机上限
P3_PoleMotor2_N_OT      :BOOL;//短路NG料盒顶升电机下限
P3_PoleMotor2_bHave		:BOOL;//短路NG料盒有料感应
P3_PoleMotor3_JogP      :BOOL;//称重和测厚NG排杆电机正转
P3_PoleMotor3_JogN      :BOOL;//称重和测厚NG排杆电机反转
P3_PoleMotor3_Reach     :BOOL;//称重和测厚NG料盒到位感应
P3_PoleMotor3_Height    :BOOL;//称重和测厚NG料盒高度感应
P3_PoleMotor3_P_OT      :BOOL;//称重和测厚NG料盒顶升电机上限
P3_PoleMotor3_N_OT      :BOOL;//称重和测厚NG料盒顶升电机下限
P3_PoleMotor3_bHave		:BOOL;//称重和测厚NG料盒有料感应
P3_PoleMotor4_JogP      :BOOL;//扫码NG排杆电机正转
P3_PoleMotor4_JogN      :BOOL;//扫码NG排杆电机反转
P3_PoleMotor4_Reach     :BOOL;//扫码NG料盒到位感应
P3_PoleMotor4_Height    :BOOL;//扫码NG料盒高度感应
P3_PoleMotor4_P_OT      :BOOL;//扫码NG料盒顶升电机上限
P3_PoleMotor4_N_OT      :BOOL;//扫码NG料盒顶升电机下限
P3_PoleMotor4_bHave		:BOOL;//扫码NG料盒有料感应
P3_ColdEmptyPress       :BOOL;//冷压空压感应
P3_HotEmptyPress        :BOOL;//冷压空压感应
P3_ColdScapegoat        :BOOL;//冷压替罪羊检测
P3_HotScapegoat         :BOOL;//冷压替罪羊检测
P3_OVenScapegoat1      :BOOL;//烤箱1替罪羊
P3_OVenScapegoat2      :BOOL;//烤箱2替罪羊
P3_OVenScapegoat3      :BOOL;//烤箱3替罪羊
P3_WeightSensor         :BOOL;//称重有料感应
P3_ThicknessSensor      :BOOL;//测厚有料感应
P3_CacheSensor          :BOOL;//缓存有料感应
P3_HotMoveOffset_X      :BOOL;//热压上料偏移检测1X
P3_HotMoveOffset_Y      :BOOL;//热压上料偏移检测2Y
P3_HotMoveOffset_Z      :BOOL;//热压上料偏移检测3Z
P3_HotOffset_L           :BOOL;//热压电芯短路测试偏移检测左   
P3_HotOffset_R           :BOOL;//热压电芯短路测试偏移检测右
P3_Ovendoorswitch1      :BOOL;//烤箱1对射感应
P3_Ovendoorswitch2      :BOOL;//烤箱2对射感应
P3_Ovendoorswitch3      :BOOL;//烤箱3对射感应
P3_Securitydoorswitch1  :BOOL;//外罩门禁1
P3_Securitydoorswitch2  :BOOL;//外罩门禁2
P3_Securitydoorswitch3  :BOOL;//外罩门禁3
P3_Securitydoorswitch4  :BOOL;//外罩门禁4
P3_Securitydoorswitch5  :BOOL;//外罩门禁5
P3_Securitydoorswitch6  :BOOL;//外罩门禁6
P3_Securitydoorswitch7  :BOOL;//外罩门禁7
P3_Securitydoorswitch8  :BOOL;//外罩门禁8
P3_Securitydoorswitch9  :BOOL;//外罩门禁9
P3_Securitydoorswitch10 :BOOL;//外罩门禁10
P3_Securitydoorswitch11 :BOOL;//外罩门禁11
P3_Securitydoorswitch12 :BOOL;//外罩门禁12
P3_Securitydoorswitch13 :BOOL;//外罩门禁13
P3_Securitydoorswitch14 :BOOL;//外罩门禁14
P3_Securitydoorswitch15 :BOOL;//外罩门禁15
P3_Securitydoorswitch16 :BOOL;//外罩门禁16
P3_ShortTest_Start      :BOOL;//短路测试测量开始
P3_ShortTest_UpperFall  :BOOL;//短路测试结果超上限
P3_ShortTest_LowerFall  :BOOL;//短路测试结果超下限
P3_ShortTest_Testing    :BOOL;// 短路测试中
P3_ShortTest_Pass       :BOOL;//短路测试OK
P3_Cold_clear           :BOOL;//冷压清零
P3_Hot_clear            :BOOL;//热压清零
P3_Tricolorlamp_Yellow  :BOOL;//后段三色灯-黄
P3_Tricolorlamp_Red		:BOOL;//后段三色灯-红
P3_Tricolorlamp_Green	:BOOL;//后段三色灯-绿
P3_Tricolorlamp_Buzzer	:BOOL;//后段三色灯-蜂鸣器

P3_InLayOffPer1:BOOL;//下料1位允许放料
P3_InLayOffPer2:BOOL;//下料2位允许放料
P3_OutSafe:BOOL;//下料位置安全
P3_OutSendFinish:BOOL;//下料放料完成

P3_Lyslgy:BOOL;//冷压上料夹电芯有无
P3_Kxslgy:BOOL;//烤箱夹电芯有无
P3_Czslgy:BOOL;//称重上料夹电芯有无
P3_Fxjgy:BOOL;//分选夹电芯有无
P3_Xljgy:BOOL;//下料夹电芯有无

P3_Oven_Power1   	:BOOL;//烤箱电源1
P3_Oven_Power2   	:BOOL;//烤箱电源2
P3_Oven_Power3   	:BOOL;//烤箱电源3
P3_Hotpress_Power   :BOOL;//热压电源

//新增
P3_IDMark:BOOL;//二维码胶Mark孔检测
P3_IDHavetape:BOOL;//二维码胶胶卷有料检测
P3_BuleHavetape:BOOL;//蓝胶胶卷有料检测
END_STRUCT
END_TYPE

// ---- P3UDTs/P3_Memory/ST_CellMemory.TcDUT
TYPE ST_CellMemory :
STRUCT
Cell      				 :BOOL;//ON、有电芯，OFF、无电芯
BlueGlue  				 :INT;//1、蓝胶OK，2、蓝胶NG
ShortTest 				 :INT;//1、短路测试OK，2、短路测试NG
Weight     				 :INT;//1、称重测试OK，2、称重测试NG
Thickness  				 :INT;//1、测厚测试OK，2、测厚测试NG
StickIDGlue_Finish :BOOL;//二维码胶贴胶完成信号

DiaphragmUnwindingTension		:	REAL	;//	隔膜放卷张力
DiaphragmUnwindingTension_max	:	REAL	;//	隔膜放卷张力-最大值
DiaphragmUnwindingTension_min	:	REAL	;//	隔膜放卷张力-最小值
DiaphragmUnwindingTension_ave	:	REAL	;//	隔膜放卷张力-平均值
DiaphragmUnwindingTension_set	:	REAL	;//	隔膜放卷张力设定值
DT_speed						:	REAL	;//	叠片速度

Overhang_Result                     :ARRAY[1..240]  OF      INT;//对齐度每一片结果
OverhandiPliesNo					:ARRAY[1..240]  OF 		INT;//返回极片层数

An_Ear_Overhang_A_C					:ARRAY[1..120]  OF		REAL	;//	正极极耳侧A/C Overhang
An_Ear_Overhang_S_CIL				:ARRAY[1..120]  OF		REAL	;//	正极极耳侧S/CIL Overhang
An_Ear_Overhang_CIL_A				:ARRAY[1..120]  OF		REAL	;//	正极极耳侧CIL/A Overhang
An_Ear_No_Overhang_A_C				:ARRAY[1..120]  OF		REAL	;//	正极非极耳侧A/C Overhang
An_Ear_No_Overhang_S_A				:ARRAY[1..120]  OF		REAL	;//	正极非极耳侧S/A Overhang
An_Ear_L_Overhang_A_C				:ARRAY[1..120]  OF		REAL	;//	正极左侧边 A/C Overhang
An_Ear_L_Overhang_S_A				:ARRAY[1..120]  OF		REAL	;//	正极左侧边 S/A Overhang
An_Ear_R_Overhang_A_C				:ARRAY[1..120]  OF		REAL	;//	正极右侧边 A/C Overhang
An_Ear_R_Overhang_S_A				:ARRAY[1..120]  OF		REAL	;//	正极右侧边 S/A Overhang

Ca_Ear_Overhang_A_C					:ARRAY[1..120]  OF		REAL	;//	负极极耳侧A/C Overhang
Ca_Ear_Overhang_S_CIL				:ARRAY[1..120]  OF		REAL	;//	负极极耳侧S/CIL Overhang
Ca_Ear_Overhang_CIL_A				:ARRAY[1..120]  OF		REAL	;//	负极极耳侧CIL/A Overhang
Ca_Ear_No_Overhang_A_C				:ARRAY[1..120]  OF		REAL	;//	负极非极耳侧A/C Overhang
Ca_Ear_No_Overhang_S_A				:ARRAY[1..120]  OF		REAL	;//	负极非极耳侧S/A Overhang
Ca_Ear_L_Overhang_A_C				:ARRAY[1..120]  OF		REAL	;//	负极左侧边 A/C Overhang
Ca_Ear_L_Overhang_S_A				:ARRAY[1..120]  OF		REAL	;//	负极左侧边 S/A Overhang
Ca_Ear_R_Overhang_A_C				:ARRAY[1..120]  OF		REAL	;//	负极右侧边 A/C Overhang
Ca_Ear_R_Overhang_S_A				:ARRAY[1..120]  OF		REAL	;//	负极右侧边 S/A Overhang


An_PoleOverhandX2					:ARRAY[1..120]  OF		REAL	;//	正极片  极片与隔膜X2
An_PoleOverhandY2					:ARRAY[1..120]  OF		REAL	;//	正极片  极片与隔膜Y2
An_PoleOverhandX3					:ARRAY[1..120]  OF		REAL	;//	正极片  极片与隔膜X3
An_PoleOverhandY3					:ARRAY[1..120]  OF		REAL	;//	正极片  极片与隔膜Y3
An_AnCaOverhandX2					:ARRAY[1..120]  OF		REAL	;//	正极片  正极到负极X2
An_AnCaOverhandY2					:ARRAY[1..120]  OF		REAL	;//	正极片  正极到负极Y2
An_AnCaOverhandX3					:ARRAY[1..120]  OF		REAL	;//	正极片  正极到负极X3
An_AnCaOverhandY3					:ARRAY[1..120]  OF		REAL	;//	正极片  正极到负极Y3
An_AddOverhangX2					:		REAL	;//	正极片  极片整体对齐度X2
An_AddOverhangY2					:		REAL	;//	正极片  极片整体对齐度Y2
An_AddOverhangX3					:		REAL	;//	正极片  极片整体对齐度X3
An_AddOverhangY3					:		REAL	;//	正极片  极片整体对齐度Y3


Ca_PoleOverhandX2					:ARRAY[1..120]  OF		REAL	;//	负极片  极片与隔膜X2
Ca_PoleOverhandY2					:ARRAY[1..120]  OF		REAL	;//	负极片  极片与隔膜Y2
Ca_PoleOverhandX3					:ARRAY[1..120]  OF		REAL	;//	负极片  极片与隔膜X3
Ca_PoleOverhandY3					:ARRAY[1..120]  OF		REAL	;//	负极片  极片与隔膜Y3
Ca_AnCaOverhandX2					:ARRAY[1..120]  OF		REAL	;//	负极片  正极到负极X2
Ca_AnCaOverhandY2					:ARRAY[1..120]  OF		REAL	;//	负极片  正极到负极Y2
Ca_AnCaOverhandX3					:ARRAY[1..120]  OF		REAL	;//	负极片  正极到负极X3
Ca_AnCaOverhandY3					:ARRAY[1..120]  OF		REAL	;//	负极片  正极到负极Y3
Ca_AddOverhangX2					:		REAL	;//	负极片  极片整体对齐度X2
Ca_AddOverhangY2					:		REAL	;//	负极片  极片整体对齐度Y2
Ca_AddOverhangX3					:		REAL	;//	负极片  极片整体对齐度X3
Ca_AddOverhangY3					:		REAL	;//	负极片  极片整体对齐度Y3

Sequeue								:ARRAY[1..120]  OF		REAL     ;//系号（无意义）

An_Cell_Overhang				:	REAL	;//	正极片整体对齐度-极耳侧
An_Cell_Overhang_No				:	REAL	;//	正极片整体对齐度-非极耳侧
An_Cell_Overhang_L				:	REAL	;//	正极片整体对齐度-左侧边
An_Cell_Overhang_R				:	REAL	;//	正极片整体对齐度-右侧边
Ca_Cell_Overhang				:	REAL	;//	负极片整体对齐度-极耳侧
Ca_Cell_Overhang_No				:	REAL	;//	负极片整体对齐度-非极耳侧
Ca_Cell_Overhang_L				:	REAL	;//	负极片整体对齐度-左侧边
Ca_Cell_Overhang_R				:	REAL	;//	负极片整体对齐度-右侧边

An_Quantity              :UINT;//正极叠片层数
Ca_Quantity              :UINT;//负极叠片层数
Machine_No				 :STRING;//叠片机编号
DT_station_No			 :STRING;//叠台工位编号*
Cleanliness_Time		 :INT;//洁净度测试时间
Cleanliness				 :INT;//洁净度
Hough     				 :INT;//(叠片台CCD综合评定结果 /对齐度) 1、对齐度OK，2、对齐度NG
ScanCode   				 :INT;//1、扫贴胶码OK,2、贴胶扫码NG
ColdPress_SV			 :REAL;//冷压压力设定值
ColdPress_PV			 :REAL;//冷压压力实际值
ColdPress_SV_H			 :REAL;//冷压压力设定值上限
ColdPress_SV_L			 :REAL;//冷压压力设定值下限
ColdPress_Time			 :UINT;//冷压时间设定值
OvenTemp_SV				 :REAL;//预热温度设定值

OvenTemp_PV				 :REAL;//预热温度实际值

OvenTemp_H				 :REAL;//预热温度上限
OvenTemp_L				 :REAL;//预热温度下限
OvenTemp_Time			 :INT;//预热时间(单位：S)

OvenShift_Time			:UDINT;//预热转移时间
OvenShift_NG_T			:BOOL;//转移时间NG


HotTemp_SV				 :REAL;//热压温度设定值

HotTemp_PV				 :REAL;//热压温度实际值

HotTemp_H				 :REAL;//热压温度设定上限
HotTemp_L				 :REAL;//热压温度设定下限
HotPress_SV			     :REAL;//热压压力设定值
HotPress_PV			     :REAL;//热压压力实际值
HotPress_SV_H			 :REAL;//热压压力设定值上限
HotPress_SV_L			 :REAL;//热压压力设定值下限
HotPress_Time			 :UINT;//热压时间设定值

Hipot_V					 :REAL;//hopot测试电压
Hipot_Time				 :REAL;//hopot测试时间
Hipot_R					 :REAL;//hopot测试电阻阻值
Hipot2_R				 :REAL;//hopot二次测试电阻阻值
Cell_Thickness       	 :REAL;//电芯厚度
Cell_weight              :REAL;//电芯重量
Operator_name			 :STRING;//作业员
Facility_NO				 :STRING;//设备机台号
Put_Time				 :STRING;//投入时间
Out_Time				 :STRING;//产出时间
Cell_number              :STRING;//电芯条码
Cell_number1             :STRING;//冷压电芯条码
Cell_cold_result		 :BOOL;//冷压上料MES判断结果
Cell_cold_result1		 :BOOL;//校对数据MES判断结果
Cell_cold_result2		 :BOOL;//上传热压数据MES判断结果
Cell_all_result			 :BOOL;//MES和本地总判定结果

Cell_CCD_No				 :STRING;//CCD电芯编号
Process_name			 :STRING;//工序名
Classes					 :STRING;//班次
Cell_result				 :INT;//综合评定结果;1、OK 2、短路NG 3、测厚NG 4、扫码NG
An_stuff_No				 :STRING;//正极极卷号，1、同卷，2、异卷
Ca_stuff_No				 :STRING;//负极极卷号，1、同卷，2、异卷
Diaphragm_No			 :STRING;//隔膜批次
QR_code_No				 :STRING;//二维码批次
Glue_No					 :STRING;//收尾胶批次

An_MQ_Slice				 :ARRAY[1..120]  OF		ST_BeltData;//正极模切极片数据
Ca_MQ_Slice				 :ARRAY[1..120]  OF		ST_BeltData;//负极模切极片数据
Overhang_TF 			 :BOOL;//对齐度NG踢废信号

core_final_result                       :  STRING(1024)  ;   // 电芯最终结果  
DP_PLC_Evaluation_result                :  STRING(1024)  ;   // 叠片PLC评定结果  
DP_MES_Evaluation_result                :  STRING(1024)  ;   // 叠片MES接口评定结果  
RY_PLC_Evaluation_result                :  STRING(1024)  ;   // 热压PLC评定结果
RY_MES_Evaluation_result                :  STRING(1024)  ;   // 热压MES接口评定结果
DP_NG_particulars                       :  STRING(1024)  ;   // 叠片NG详情    
RY_NG_particulars                       :  STRING(1024)  ;   //  热压NG详情 

DP_Internal_decision_details            :  STRING(1024)  ;   // 叠片内部判定详情
DP_External_decision_details            :  STRING(1024)  ;   // 叠片外部判定详情 
RY_Internal_decision_details            :  STRING(1024)  ;   // 热压内部判定详情 
RY_External_decision_details            :  STRING(1024)  ;   // 热压外部判定详情

//PC写给PLC的-----先下发给叠台，叠台再和模切做通讯
PostiveCode			:STRING(49);//正极条码		
NegativeCode			:STRING(49);//负极条码		
Station_Code			:STRING(49);//叠台隔膜条码		
Station_BlueCode		:STRING(49);//叠台蓝胶条码		
P3CellCode			:STRING(49);//后段二维码胶条码	
P3BlueCode			:STRING(49);//后段蓝胶条码		

ColdPress_PVTime			 :UINT;//冷压时间实际值
OvenTemp_NO              :INT;// 预热工位号
OvenTemp_PVTime			 :UDINT;//预热实际时间
HotPress_PVTime			 :UINT;//热压时间实际值

DiaphragmUnwindingTension2		:ARRAY[1..240]  OF	REAL	;//	隔膜放卷张力每一片
DTDebugMode           :BOOL;//叠台调试模式    

//20240417WCZ
LYDLineinitPos	 : REAL ;// 	左压刀开合初始位
LYDLineOpenPos 	 : REAL ;// 	左压刀开合张开位
LYDLinepressL 	 : REAL ;// 	左压刀开合压隔膜长度
RYDLineinitPos	 : REAL ;// 	右压刀开合初始位
RYDLineOpenPos 	 : REAL ;// 	右压刀开合张开位
RYDLinepressL 	 : REAL ;// 	右压刀开合压隔膜长度
LYDUpDowninitPos	 : REAL ;// 	左压刀升降初始位
LYDUpDownOpenPos 	 : REAL ;// 	左压刀升降张开位
LYDUpDownOpenH	 : REAL ;// 	左压刀升降张开高度
LYDUpDownKnifeH	 : REAL ;// 	左压刀升降抽刀高度
RYDUpDowninitPos 	 : REAL ;// 	右压刀升降初始位
RYDUpDownOpenPos 	 : REAL ;// 	右压刀升降张开位
RYDUpDownOpenH	 : REAL ;// 	右压刀升降张开高度
RYDUpDownKnifeH	 : REAL ;// 	右压刀升降抽刀高度
DTandescendh	 : REAL ;// 	叠台正极片下降高度
DTcadescendh	 : REAL ;// 	叠台负极片下降高度
Shortpress	 : REAL ;// 	短路测试压力（Kg)
coldActPos	 : REAL ;// 	冷压板实际位置
HeatActPos	 : REAL ;// 	热压板实际位置
Chipdata   :ARRAY[1..240]  OF Mes2 ;//极片数据                               	
END_STRUCT
END_TYPE

// ---- P3UDTs/P3_Name/ST_MemoryName.TcDUT
TYPE ST_MemoryName :
STRUCT

Dietai1          :INT:=1;//1号叠台电芯记忆
Weijuan1         :INT:=2;//1号尾卷电芯记忆
Gluing1          :INT:=3;//1号贴胶电芯记忆
Dietai2          :INT:=4;//2号叠台电芯记忆
Weijuan2         :INT:=5;//2号尾卷电芯记忆
Gluing2          :INT:=6;//2号贴胶电芯记忆
Dietai3          :INT:=7;//3号叠台电芯记忆
Weijuan3         :INT:=8;//3号尾卷电芯记忆
Gluing3          :INT:=9;//3号贴胶电芯记忆
ColdpressClip    :INT:=10;//冷压上料夹子电芯记忆
Coldpress        :INT:=11;//冷压电芯记忆
OvenMoveClip1    :INT:=12;//冷压下料到烤箱时夹子电芯记忆
Oven_M1          :INT:=13;//烤箱位置1的电芯记忆
Oven_M2          :INT:=14;//烤箱位置2的电芯记忆
Oven_M3          :INT:=15;//烤箱位置3的电芯记忆
Oven_M4          :INT:=16;//烤箱位置4的电芯记忆
Oven_M5          :INT:=17;//烤箱位置5的电芯记忆
Oven_M6          :INT:=18;//烤箱位置6的电芯记忆
Oven_M7          :INT:=19;//烤箱位置7的电芯记忆
Oven_M8          :INT:=20;//烤箱位置8的电芯记忆
Oven_M9          :INT:=21;//烤箱位置9的电芯记忆
Oven_M10         :INT:=22;//烤箱位置10的电芯记忆
Oven_M11         :INT:=23;//烤箱位置11的电芯记忆
Oven_M12         :INT:=24;//烤箱位置12的电芯记忆
Oven_M13         :INT:=25;//烤箱位置13的电芯记忆
Oven_M14         :INT:=26;//烤箱位置14的电芯记忆
Oven_M15         :INT:=27;//烤箱位置15的电芯记忆
Oven_M16         :INT:=28;//烤箱位置16的电芯记忆
Oven_M17         :INT:=29;//烤箱位置17的电芯记忆
Oven_M18         :INT:=30;//烤箱位置18的电芯记忆
Oven_M19         :INT:=31;//烤箱位置19的电芯记忆
Oven_M20         :INT:=32;//烤箱位置20的电芯记忆
Oven_M21         :INT:=33;//烤箱位置21的电芯记忆
Oven_M22         :INT:=34;//烤箱位置22的电芯记忆
Oven_M23         :INT:=35;//烤箱位置23的电芯记忆
Oven_M24         :INT:=36;//烤箱位置24的电芯记忆
Oven_M25         :INT:=37;//烤箱位置25的电芯记忆
Oven_M26         :INT:=38;//烤箱位置26的电芯记忆
Oven_M27         :INT:=39;//烤箱位置27的电芯记忆
Oven_M28         :INT:=40;//烤箱位置28的电芯记忆
Oven_M29         :INT:=41;//烤箱位置29的电芯记忆
Oven_M30         :INT:=42;//烤箱位置30的电芯记忆
Oven_M31         :INT:=43;//烤箱位置31的电芯记忆
Oven_M32         :INT:=44;//烤箱位置32的电芯记忆
Oven_M33         :INT:=45;//烤箱位置33的电芯记忆
Oven_M34         :INT:=46;//烤箱位置34的电芯记忆
Oven_M35         :INT:=47;//烤箱位置35的电芯记忆
Oven_M36         :INT:=48;//烤箱位置36的电芯记忆
Oven_M37         :INT:=49;//烤箱位置37的电芯记忆
Oven_M38         :INT:=50;//烤箱位置38的电芯记忆
Oven_M39         :INT:=51;//烤箱位置39的电芯记忆
Oven_M40         :INT:=52;//烤箱位置40的电芯记忆
Oven_M41         :INT:=53;//烤箱位置41的电芯记忆
Oven_M42         :INT:=54;//烤箱位置42的电芯记忆
OvenMoveClip2    :INT:=55;//烤箱下料到热压时烤箱夹子电芯记忆
Hotpress         :INT:=56;//热压电芯记忆
WeightClip       :INT:=57;//称重上料夹子电芯记忆
Weight           :INT:=58;//称重平台电芯记忆
SortClip1        :INT:=59;//电芯分选夹子去取称重平台时夹子的电芯记忆
Thickness        :INT:=60;//测厚平台上的电芯记忆
SortClip2        :INT:=61;//电芯分选夹子去取测厚平台时夹子的电芯记忆
BlankingPlatform :INT:=62;//下料辅助平台上的电芯记忆
BlankingClip     :INT:=63;//下料夹子的电芯记忆


END_STRUCT
END_TYPE

// ---- P3UDTs/P3_Name/ST_P3AxisName.TcDUT
TYPE ST_P3AxisName :
STRUCT
P3M1_ColdpreLine	         :INT:=160; //	P3_M1冷压上料夹平移, 1、初始位，2、贴胶1位，3、贴胶2位，4、贴胶3位，5、冷压位，6、排NG料1位，7、排NG料2位
P3M1_ColdpreRetracting	     :INT:=161;	//	P3_M1冷压上料夹进退  1、初始位，2、贴胶1位，3、贴胶2位，4、贴胶3位，5、冷压位，6、排NG料位
P3M1_ColdpreWhirling	     :INT:=162;	//	P3_M1冷压上料夹旋转  1、初始位，2、贴胶1位，3、贴胶2位，4、贴胶3位，5、冷压位，6、排NG料位
P3M1_ColdpreUpDown	         :INT:=163; //	P3_M1冷压上料夹升降  1、初始位，2、贴胶1位，3、贴胶2位，4、贴胶3位，5、冷压位，6、排NG料位  7、贴胶1辅助位  8、贴胶2辅助位  9、贴胶3辅助位  10、冷压辅助位
P3M1_ColdpreSupPlateLine	 :INT:=164;	//	P3_M1冷压托板开合    1、初始位，2、张开位
P3M1_ColdpreActuated	     :INT:=165;	//	P3_M1冷压驱动        1、初始位, 2、电芯位
P3_M2_OvenCarrying	         :INT:=166;	//	P3_M2烤箱上料夹搬运 43、初始位，44、冷压位，45、热压位，1-42、烤箱位，46、扫码位，47、贴二维码胶位
P3_M2_OvenRetracting	     :INT:=167;	//	P3_M2烤箱上料夹进退 43、初始位，44、冷压位，45、热压位，1-42、烤箱位，46、扫码位和贴二维码胶位
P3_M2_OvenUpDown	         :INT:=168;	//	P3_M2烤箱上料夹升降 43、初始位，44、冷压位，45、热压位，1-42、烤箱位，46、扫码位和贴二维码胶位 48、热压辅助位 49、冷压辅助位
P3_M3_HotPressingLine	     :INT:=169;	//	P3_M3热压托板开合    1、初始位，2、张开位
P3_M3_HotPressingActuated	 :INT:=170;	//	P3_M3热压驱动        1、初始位，2、电芯位
P3_M4_WeighLine	             :INT:=171;	//	P3_M4称重上料夹平移  1、初始位，2、热压位，3、称重位   4、避让位(可旋转)
P3_M4_WeighUpDown	         :INT:=172;	//	P3_M4称重上料夹升降  1、初始位，2、热压位，3、称重位  4、热压辅助位   5、称重辅助位
P3_M4_WeighWhirling	         :INT:=173;	//	P3_M4称重上料夹旋转  1、初始位，2、热压位，3、称重位
P3_M4_SortingoutCarrying	 :INT:=174;	//	P3_M4电芯分选夹搬运  1、初始位，2、称重位，3、测厚位，4、放料位，5、1号料盒短路对齐度NG位，6、2号料盒厚度烘烤NG位，7、3号料盒扫码称重mesNG位
P3_M4_SortingoutUpDown	     :INT:=175;	//	P3_M4电芯分选夹升降  1、初始位，2、称重位，3、测厚位，4、放料位，5、短路NG位，6、称重和测厚NG位，7扫码NG位,8称重辅助位，9测厚辅助位
P3_M4_OffloadingCarrying	 :INT:=176;	//	P3_M4电芯下料夹搬运  1、初始位，2、取料位，3、下料位1  4、下料位2
P3_M4_OffloadingUpDown	     :INT:=177;	//	P3_M4电芯下料夹升降  1、初始位，2、取料位，3、下料位, 4、取料下降位 5、等待高度 6、下料下降位
P3_TapeAdvance				:INT:=178;	//	P3_M3贴胶头进退1=初始位,2=取胶位,3=非极耳侧贴胶位,4=贴胶等待位,5=极耳侧贴胶位
P3_TapeTranslation			:INT:=179;	//	P3_M3贴胶平移1=贴胶1位，2=贴胶2位，3=贴胶3位，4=贴胶4位，5=贴胶5位，6=贴胶6位，7=下料位，,8=初始位

//新增
P3_IDPut							:INT:=180;//二维码胶拉胶		1:初始位  2:取胶位  3:拉胶位  4:切胶最小位 5:切胶最大位	6,Mark孔后定长 7,NG位
P3_IDLift							:INT:=181;//二维码胶升降		1:初始位  2:取胶位  3:贴胶位  4:避让位  5:NG位

END_STRUCT
END_TYPE

// ---- P3UDTs/P3_Name/ST_P3CylinderName.TcDUT
TYPE ST_P3CylinderName :
STRUCT
P3ColdPressClip	:INT:=230;	//	P3	冷压上料夹气缸
P3ColdPressTensed	:INT:=231;	//	P3	冷压麦拉张紧气缸
P3OvenMoveClip	:INT:=232;	//	P3	烤箱上料夹气缸
P3Oven1	:INT:=233;	//	P3	1_1烤箱托板气缸
P3Oven2	:INT:=234;	//	P3	1_2烤箱托板气缸
P3Oven3	:INT:=235;	//	P3	1_3烤箱托板气缸
P3Oven4	:INT:=236;	//	P3	1_4烤箱托板气缸
P3Oven5	:INT:=237;	//	P3	1_5烤箱托板气缸
P3Oven6	:INT:=238;	//	P3	1_6烤箱托板气缸
P3Oven7	:INT:=239;	//	P3	1_7烤箱托板气缸
P3Oven8	:INT:=240;	//	P3	2_1烤箱托板气缸
P3Oven9	:INT:=241;	//	P3	2_2烤箱托板气缸
P3Oven10	:INT:=242;	//	P3	2_3烤箱托板气缸
P3Oven11	:INT:=243;	//	P3	2_4烤箱托板气缸
P3Oven12	:INT:=244;	//	P3	2_5烤箱托板气缸
P3Oven13	:INT:=245;	//	P3	2_6烤箱托板气缸
P3Oven14	:INT:=246;	//	P3	2_7烤箱托板气缸
P3Oven15	:INT:=247;	//	P3	3_1烤箱托板气缸
P3Oven16	:INT:=248;	//	P3	3_2烤箱托板气缸
P3Oven17	:INT:=249;	//	P3	3_3烤箱托板气缸
P3Oven18	:INT:=250;	//	P3	3_4烤箱托板气缸
P3Oven19	:INT:=251;	//	P3	3_5烤箱托板气缸
P3Oven20	:INT:=252;	//	P3	3_6烤箱托板气缸
P3Oven21	:INT:=253;	//	P3	3_7烤箱托板气缸
P3HotPressTensed	:INT:=254;	//	P3	热压麦拉张紧气缸
P3ShortTest	:INT:=255;	//	P3	短路测试夹气缸
P3WeightFeedingClamp	:INT:=256;	//	P3	称重上料夹气缸
P3ThicknessMeasuringSwitch	:INT:=257;	//	P3	测厚台切换气缸
P3ThicknessSupport	:INT:=258;	//	P3	测厚台托板气缸
P3ThicknessPressure	:INT:=259;	//	P3	测厚台压板气缸
P3SortClamp	:INT:=260;	//	P3	电芯分选夹开合气缸
P3SortLifting	:INT:=261;	//	P3	电芯分选夹升降气缸
P3SortRotate	:INT:=262;	//	P3	电芯分选夹旋转气缸
P3BlankingClamp	:INT:=263;	//	P3	电芯下料夹开合气缸
P3BlankingLifting	:INT:=264;	//	P3	电芯下料夹升降气缸
P3BlankingRotate	:INT:=265;	//	P3	电芯下料夹旋转气缸
P3BoxLock1_NG	:INT:=266;	//	P3	电芯NG1料盒锁定气缸
P3BoxLock2_NG	:INT:=267;	//	P3	电芯NG2料盒锁定气缸
P3BoxLock3_NG	:INT:=268;	//	P3	电芯NG3料盒锁定气缸
(*P3Cold_Clamp	   :INT:=269;  //  P3  冷压辅助上料开合气缸
P3Cold_Tensed	   :INT:=270;  //  P3  冷压辅助上料夹紧气缸
P3Cold_Retracting  :INT:=271;  //  P3  冷压辅助上料进退气缸
P3Cold_Lifting	   :INT:=272;  //  P3  冷压辅助上料升降气缸*)

//新增

//新增

P3CellPush:INT:=269;//电芯压紧气缸
P3CellAdvance:INT:=270;//电芯平移气缸
P3TapePush:INT:=271;//贴胶头夹紧气缸
P3TapePull:INT:=272;//拉带夹紧气缸
P3TapeLift:INT:=273;//拉带升降气缸
P3TapeCut:INT:=274;//切胶气缸
P3GluePush:INT:=275;//压胶气缸
P3TapeBuffer:INT:=276;//贴胶缓存气缸
P3TapeSpin:INT:=277;//流水线下料旋转气缸
P3TapeVacuo:INT:=278;//贴胶头真空
P3WgightUP:INT:=279;//称重上料夹夹电芯气缸
P3SortPush:INT:=280;//电芯分选夹夹电芯气缸
P3ColdBlow:INT:=281;//冷压吹气
P3HotBlow:INT:=282;//热压吹气
P3CellPushSpin:INT:=283;//电芯旋转定位气缸
P3CellSpin:INT:=284;//电芯旋转气缸



//新增
P3_GlueExtend:INT:=285;//二维码蹬胶气缸
P3_GluePress:INT:=286;	//二维码压胶气缸
P3_GlueCut:INT:=287;	//二维码切胶气缸
P3_GluePull:INT:=288;	//二维码拉胶气缸
P3_GlueVacuum:INT:=289;//	二维码贴胶吸盘真空 ON真空 OFF破真空

END_STRUCT
END_TYPE

// ---- P3UDTs/P3_Name/ST_P3ElectValveName.TcDUT
TYPE ST_P3ElectValveName :
STRUCT
		
END_STRUCT
END_TYPE

// ---- P3UDTs/P3_Name/ST_TempName.TcDUT
TYPE ST_TempName :   //  整机纠偏名称
STRUCT
	
//烤箱1加热板				
P3_PoleBoard1_1	:INT:=1;	//箱烤	1	上加热板1
P3_PoleBoard1_2	:INT:=2;	//箱烤	1	上加热板2
P3_PoleBoard1_3	:INT:=3;	//箱烤	1	下加热板1
P3_PoleBoard1_4	:INT:=4;	//箱烤	1	下加热板2
//烤箱2加热板				
P3_PoleBoard2_1	:INT:=5;	//箱烤	2	上加热板1
P3_PoleBoard2_2	:INT:=6;	//箱烤	2	上加热板2
P3_PoleBoard2_3	:INT:=7;	//箱烤	2	下加热板1
P3_PoleBoard2_4	:INT:=8;	//箱烤	2	下加热板2
//烤箱3加热板				
P3_PoleBoard3_1	:INT:=9;	//箱烤	3	上加热板1
P3_PoleBoard3_2	:INT:=10;	//箱烤	3	上加热板2
P3_PoleBoard3_3	:INT:=11;	//箱烤	3	下加热板1
P3_PoleBoard3_4	:INT:=12;	//箱烤	3	下加热板2
//烤箱4加热板				
P3_PoleBoard4_1	:INT:=13;	//箱烤	4	上加热板1
P3_PoleBoard4_2	:INT:=14;	//箱烤	4	上加热板2
P3_PoleBoard4_3	:INT:=15;	//箱烤	4	下加热板1
P3_PoleBoard4_4	:INT:=16;	//箱烤	4	下加热板2
//烤箱5加热板				
P3_PoleBoard5_1	:INT:=17;	//箱烤	5	上加热板1
P3_PoleBoard5_2	:INT:=18;	//箱烤	5	上加热板2
P3_PoleBoard5_3	:INT:=19;	//箱烤	5	下加热板1
P3_PoleBoard5_4	:INT:=20;	//箱烤	5	下加热板2
//烤箱6加热板				
P3_PoleBoard6_1	:INT:=21;	//箱烤	6	上加热板1
P3_PoleBoard6_2	:INT:=22;	//箱烤	6	上加热板2
P3_PoleBoard6_3	:INT:=23;	//箱烤	6	下加热板1
P3_PoleBoard6_4	:INT:=24;	//箱烤	6	下加热板2
//烤箱7加热板				
P3_PoleBoard7_1	:INT:=25;	//箱烤	7	上加热板1
P3_PoleBoard7_2	:INT:=26;	//箱烤	7	上加热板2
P3_PoleBoard7_3	:INT:=27;	//箱烤	7	下加热板1
P3_PoleBoard7_4	:INT:=28;	//箱烤	7	下加热板2
//烤箱8加热板				
P3_PoleBoard8_1	:INT:=33;	//箱烤	8	上加热板1
P3_PoleBoard8_2	:INT:=34;	//箱烤	8	上加热板2
P3_PoleBoard8_3	:INT:=35;	//箱烤	8	下加热板1
P3_PoleBoard8_4	:INT:=36;	//箱烤	8	下加热板2
//烤箱9加热板				
P3_PoleBoard9_1	:INT:=37;	//箱烤	9	上加热板1
P3_PoleBoard9_2	:INT:=38;	//箱烤	9	上加热板2
P3_PoleBoard9_3	:INT:=39;	//箱烤	9	下加热板1
P3_PoleBoard9_4	:INT:=40;	//箱烤	9	下加热板2
//烤箱10加热板				
P3_PoleBoard10_1	:INT:=41;	//箱烤	10	上加热板1
P3_PoleBoard10_2	:INT:=42;	//箱烤	10	上加热板2
P3_PoleBoard10_3	:INT:=43;	//箱烤	10	下加热板1
P3_PoleBoard10_4	:INT:=44;	//箱烤	10	下加热板2
//烤箱11加热板				
P3_PoleBoard11_1	:INT:=45;	//箱烤	11	上加热板1
P3_PoleBoard11_2	:INT:=46;	//箱烤	11	上加热板2
P3_PoleBoard11_3	:INT:=47;	//箱烤	11	下加热板1
P3_PoleBoard11_4	:INT:=48;	//箱烤	11	下加热板2
//烤箱12加热板				
P3_PoleBoard12_1	:INT:=49;	//箱烤	12	上加热板1
P3_PoleBoard12_2	:INT:=50;	//箱烤	12	上加热板2
P3_PoleBoard12_3	:INT:=51;	//箱烤	12	下加热板1
P3_PoleBoard12_4	:INT:=52;	//箱烤	12	下加热板2
//烤箱13加热板				
P3_PoleBoard13_1	:INT:=53;	//箱烤	13	上加热板1
P3_PoleBoard13_2	:INT:=54;	//箱烤	13	上加热板2
P3_PoleBoard13_3	:INT:=55;	//箱烤	13	下加热板1
P3_PoleBoard13_4	:INT:=56;	//箱烤	13	下加热板2
//烤箱14加热板				
P3_PoleBoard14_1	:INT:=57;	//箱烤	14	上加热板1
P3_PoleBoard14_2	:INT:=58;	//箱烤	14	上加热板2
P3_PoleBoard14_3	:INT:=59;	//箱烤	14	下加热板1
P3_PoleBoard14_4	:INT:=60;	//箱烤	14	下加热板2
//烤箱15加热板				
P3_PoleBoard15_1	:INT:=65;	//箱烤	15	上加热板1
P3_PoleBoard15_2	:INT:=66;	//箱烤	15	上加热板2
P3_PoleBoard15_3	:INT:=67;	//箱烤	15	下加热板1
P3_PoleBoard15_4	:INT:=68;	//箱烤	15	下加热板2
//烤箱16加热板				
P3_PoleBoard16_1	:INT:=69;	//箱烤	16	上加热板1
P3_PoleBoard16_2	:INT:=70;	//箱烤	16	上加热板2
P3_PoleBoard16_3	:INT:=71;	//箱烤	16	下加热板1
P3_PoleBoard16_4	:INT:=72;	//箱烤	16	下加热板2
//烤箱17加热板				
P3_PoleBoard17_1	:INT:=73;	//箱烤	17	上加热板1
P3_PoleBoard17_2	:INT:=74;	//箱烤	17	上加热板2
P3_PoleBoard17_3	:INT:=75;	//箱烤	17	下加热板1
P3_PoleBoard17_4	:INT:=76;	//箱烤	17	下加热板2
//烤箱18加热板				
P3_PoleBoard18_1	:INT:=77;	//箱烤	18	上加热板1
P3_PoleBoard18_2	:INT:=78;	//箱烤	18	上加热板2
P3_PoleBoard18_3	:INT:=79;	//箱烤	18	下加热板1
P3_PoleBoard18_4	:INT:=80;	//箱烤	18	下加热板2
//烤箱19加热板				
P3_PoleBoard19_1	:INT:=81;	//箱烤	19	上加热板1
P3_PoleBoard19_2	:INT:=82;	//箱烤	19	上加热板2
P3_PoleBoard19_3	:INT:=83;	//箱烤	19	下加热板1
P3_PoleBoard19_4	:INT:=84;	//箱烤	19	下加热板2
//烤箱20加热板				
P3_PoleBoard20_1	:INT:=85;	//箱烤	20	上加热板1
P3_PoleBoard20_2	:INT:=86;	//箱烤	20	上加热板2
P3_PoleBoard20_3	:INT:=87;	//箱烤	20	下加热板1
P3_PoleBoard20_4	:INT:=88;	//箱烤	20	下加热板2
//烤箱21加热板				
P3_PoleBoard21_1	:INT:=89;	//箱烤	21	上加热板1
P3_PoleBoard21_2	:INT:=90;	//箱烤	21	上加热板2
P3_PoleBoard21_3	:INT:=91;	//箱烤	21	下加热板1
P3_PoleBoard21_4	:INT:=92;	//箱烤	21	下加热板2
//热压加热板				
P3_HotpressBoard1	:INT:=93;		//热压加热板上板	
P3_HotpressBoard2	:INT:=94;		//热压加热板下板	


END_STRUCT
END_TYPE

// ---- P3UDTs/P3_par/P3_Par.TcDUT
TYPE P3_Par :
STRUCT
	Oven_Shijian:INT;// 烤箱烘烤时间
	CleanTimeHMIHour1:INT;//白班第一次清洁时间Hour
	CleanTimeHMIMin1:INT;//白班第一次清洁时间Min
	CleanTimeHMIHour2:INT;//白班第二次清洁时间Hour
	CleanTimeHMIMin2:INT;//白班第二次清洁时间Min
	CleanTimeHMIHour3:INT;//夜班第一次清洁时间Hour
	CleanTimeHMIMin3:INT;//夜班第一次清洁时间Min
	CleanTimeHMIHour4:INT;//夜班第二次清洁时间Hour
	CleanTimeHMIMin4:INT;//夜班第二次清洁时间Ming
	P3_Thickness_HMIStuas:INT;//记忆测厚电芯状态
	P3_Thickness_HMIThick:REAL;//记忆测厚电芯厚度
	P3_Press_SV: ARRAY [1..2] OF REAL;//设定压力值
	P3_AD_Press: ARRAY [1..2] OF REAL;// 压力模拟量
	P3_Press_Time: ARRAY [1..2] OF TIME;// 保持压力时间
    P3_Press_DeadZone :ARRAY[1..2] OF REAL;//压力死区范围
    P3_Press_Fast_xs:  ARRAY[1..2] OF REAL;//快速系数
    P3_Press_Slow_xs:  ARRAY[1..2] OF REAL;//慢速系数

END_STRUCT
END_TYPE

// ---- P3UDTs/P3_par/User2_Par.TcDUT
TYPE User2_Par :
STRUCT




     iTest                                   :INT;
///////////////////////////////////////////////////////中转变量/////////////////////////////////////////////////////////////////////////////////////////////////
	fSavePositionBias:ARRAY[1..12] OF LREAL;(*写入软限位的值*)
	HMI_Button:ARRAY[1..12]OF  BOOL;//ADS软限位开关
	Shield          :ARRAY[1..99] OF BOOL;//屏蔽功能按钮，1、屏蔽短路测试 2、屏蔽称重测试 3、屏蔽测厚测试  4、扫码屏蔽 5、上位机屏蔽 6、短路测试复测  7、冷压正常流程 20,分选夹旋转选择按钮，true不旋转，false旋转；OK  8：MES条码校验 9：二维码胶条码重新校验 10：蓝胶条码重新校验 11:1号叠台首检模式 12:2号叠台首检模式 13:3号叠台首检模式
	Oven_Shield          :ARRAY[1..21] OF BOOL;//烤箱屏蔽OK
	LateBlanking_motor :BOOL;//后段电机条件屏蔽OK
	Cold_par                :ST_TorqueMotion;//OK
	Hot_par                :ST_TorqueMotion;//OK
	Oven_finish: ARRAY [1..42] OF BOOL;// 烤箱烘烤时间完成信号  //
	Oven_Finish_Time :ARRAY[1..42] OF UDINT;//烤箱烘烤完成后计数时间//OK
	Oven_cell: ARRAY [1..42] OF BOOL;//烤箱电芯记忆
	V: INT ;// 烤箱上料记忆辅助计数
	W: INT;// 烤箱下料记忆辅助计数
	B_OVEN :BOOL;//屏蔽烤箱
	Thick_Par :REAL;//测厚基准
	Thick_MN	:REAL;//测厚误差范围
 	Thick_Cell_Par :REAL;//测厚电芯厚度

	Door_Forbidden :BOOL;//热压段门禁禁用
	Scan_IP :T_IPv4Addr;//扫码IP
	MQ_CaFSY_IP :T_IPv4Addr;//模切负极风速仪IP
	MQ_AnFSY_IP :T_IPv4Addr;//模切正极风速仪IP
	Cold_Position :REAL;//冷压上料辅助位

	Thick_min :REAL:=21.65;//测厚厚度最小值(标准)
	Thick_max :REAL:=22.65;//测厚厚度最大值(标准)
	Oven_Time_S :UDINT:=200;//预热转移时间超时NG限定时间
	
    Bounce_time :UDINT ;//弹窗时间
    Status_switching_time :UDINT ;//状态切换时间
    Standby_time :UDINT;//待料时间
	Oven_cell_Shield     :ARRAY[1..42] OF BOOL;//烤箱电芯屏蔽
	

		
		
		
END_STRUCT
END_TYPE

// ---- P3UDTs/P3_ShortTest/CMD_1.TcDUT
TYPE CMD_1 :
STRUCT
	RST :                   STRING:='*RST';     // 1 仪器初始化
    Start :                 STRING:=':STARt';// 2 测试开始
    Stop :                  STRING:=':STOP';// 3  测试停止
    State_Check :           STRING:=':STATe?';// 4 测试状态查询 0：停止中  1：测试中   2：放电中
	
    Measure_Check :         STRING:=':MEASure?';// 5  测量值查询
    Measure_Check2 :        STRING:=':MEASure:RESult?';// 6  测量值，判定结果查询  //1:OFF 2:NOcomp 3:DELAY 4:PASS 5:UFAIL 6:LFAIL 7:ULFA
    Measure_Clear :         STRING:=':MEASure:CLEar';// 7  测量值，判定结果清除
	
    Voltage :               STRING:=':VOLTage';// 8  测试电压设置
    Voltage_Check :         STRING:=':VOLTage?';// 9  测试电压查询 
    Voltage_Monitor :       STRING:=':MEASure:MONItor?';// 10  电压值监视
	
    Mohm_Range :            STRING:=':MOHM:RANGe';// 11  电阻量程设置(2M/20M/200M/2000M/4000M/AUTO)  
    Mohm_Range_Check :      STRING:=':MOHM:RANGe?';// 12  电阻量程查询
	
    Speed :                 STRING:=':SPEed';// 13 测量速度设置(FAST/SLOW)
    Speed_Check :           STRING:=':SPEed?';// 14 测量速度查询
	
    Timer :                 STRING:=':TIMer';// 15  测试时间设置
    Timer_Check :           STRING:=':TIMer?';// 16  测试时间查询
    Delay :                 STRING:=':DELay';// 17  响应时间设置(0为自动)
    Delay_Check :           STRING:=':DELay?';// 18  响应时间查询(0为自动)
	
    ComparatorLimit :       STRING:=':COMParator:LIMit';// 19  比较器上下限值设置（上限,下限）
    ComparatorLimit_Check : STRING:=':COMParator:LIMit?';// 20  比较器上下限值查询
    ComparatorMode :        STRING:=':COMParator:MODE';// 21  测试模式设置（CONTinue/PASSstop/FAILstop/SEQuence）  
    ComparatorMode_Check :  STRING:=':COMParator:MODE?';// 22 测试模式查询（CONTINUE/PASSSTOP/FAILSTOP/SEQUENCE）
    ComparatorBeeper :      STRING:=':COMParator:BEEPer';// 23  判定蜂鸣器设置(PASS/FAIL/OFF/END)
    ComparatorBeeper_Check :STRING:=':COMParator:BEEPer?';// 24  判定蜂鸣器查询(PASS/FAIL/OFF/END)
	
    Contact :               STRING:=':CONTactcheck';//  25  接触检查功能设置(ON/OFF)	
	Contact_Check :         STRING:=':CONTactcheck?';// 26  接触检查功能查询(ON/OFF)
    Contact_Result :        STRING:=':CONTactcheck:RESult?';// 27  接触检查结果查询(NOCHK/PASS/HFAIL/LFAIL/HLFAIL)
	
    Short :                 STRING:=':SHORtcheck';// 28  短路检查功能设置(ON/OFF)	
    Short_Check :           STRING:=':SHORtcheck?';// 29  短路检查功能查询 
    ShortTime :             STRING:=':SHORtcheck:TIME';// 30 短路检查时间设置(0:自动)
    ShortTime_Check :       STRING:=':SHORtcheck:TIME?';// 31  短路检查时间查询
    Short_Result :          STRING:=':SHORtcheck:RESult?';// 32  短路检查结果查询（NOCHK/PASS/FAIL）
	
    KeyBeeper :             STRING:=':KEY:BEEPer';// 33  按键输入蜂鸣器音设置(ON/OFF)	
    KeyBeeper_Check :       STRING:=':KEY:BEEPer?';// 34  按键输入蜂鸣器音查询
   
END_STRUCT
END_TYPE

// ---- P3UDTs/P3_ShortTest/ShortCiucitCtrl.TcDUT
TYPE ShortCiucitCtrl :
STRUCT
	ShortTestCtrl_U:ShortTestCtrl;
	ShortTestReceiveData_U:ShortTestReceiveData;
	ShortTestSendData_U:ShortTestSendData;
	ST_ReceiveTestStatus_U:ST_ReceiveTestStatus;
	ST_SendTestStatus_U:ST_SendTestStatus;
END_STRUCT
END_TYPE

// ---- P3UDTs/P3_ShortTest/ShortDataShow_1.TcDUT
TYPE ShortDataShow_1 :
STRUCT
	strState:STRING;         //0：停止中  1：测试中   2：放电中
    strResult:STRING;  //启动测试后返回结果   综合结果
	
	strMeasure :STRING;     //测量电阻值
	strMeasureState :STRING;     //1:OFF 2:NOcomp 3:DELAY 4:PASS 5:UFAIL 6:LFAIL 7:ULFAIL

	strVoltageSetValue:STRING;  //电压设定值查询
    strVoltageMonitor:STRING; //电压值监视
	
	strMohmRangeValue:STRING;//(1:2M/2:20M/3:200M/4:2000M/5:4000M/6:AUTO) 
    
	strSpeedValue:STRING ;//测量速度查询(FAST/SLOW)
	
	strTimerValue :STRING;  //测试时间查询
	strDelayValue :STRING;  //响应时间查询(0自动）
	
	strComparatorLimitSet :STRING;  //比较器上限 下限值
	strComparatorModeValue: STRING ;// 21  测试模式查询（CONTinue/PASSstop/FAILstop/SEQuence）
	strComparatorBeeperValue:    STRING;//23  判定蜂鸣器查询(PASS/FAIL/OFF/END)
	
	strContactValue :STRING;//  25  接触检查功能查询(ON/OFF)
	strContactResult :STRING;//  27  接触检查结果查询(NOCHK/PASS/HFAIL/LFAIL/HLFAIL)
	
	strShortValue:STRING;// 28  短路检查功能查询(ON/OFF)
	strShortTimeValue:  STRING;// 30 短路检查时间查询(0:自动)
	strShortResult:STRING;// 32  短路检查结果查询（NOCHK/PASS/FAIL）
	
	strKeyBeeperValue:STRING;  // 33  按键输入蜂鸣器音查询(ON/OFF)	

END_STRUCT
END_TYPE

// ---- P3UDTs/P3_ShortTest/ShortPar_1.TcDUT
TYPE ShortPar_1 :
STRUCT
	fVoltageSet: REAL;  //电压设定值

	StrMohmRangeSet:STRING; //电阻量程设置(1:2M/2:20M/3:200M/4:2000M/5:4000M/6:AUTO) 

    StrSpeedSet:STRING ;//测量速度设置(FAST/SLOW)
    
    fTimerSet:    REAL; //测试时间设置
    fDelaySet:   REAL; //响应时间设定
     
	fComparatorUpLimitSet :REAL;  //比较器上限设定
	fComparatorDownLimitSet :REAL;//比较器下限设定	
    strComparatorModeSet: STRING ;// 21  测试模式设置（CONTinue/PASSstop/FAILstop/SEQuence）
	
	strComparatorBeeperSet:    STRING;//23  判定蜂鸣器设置(PASS/FAIL/OFF/END)
	
	strContactSet :STRING;//  25  接触检查功能设置(ON/OFF)	

	strShortSet:STRING;// 28  短路检查功能设置(ON/OFF)
	
	fShortTimeSet:  REAL;// 30 短路检查时间设置(0:自动)
	
	
	strKeyBeeperSet:STRING;  // 33  按键输入蜂鸣器音设置(ON/OFF)	
	
	
END_STRUCT
END_TYPE

// ---- P3UDTs/P3_ShortTest/ShortTestCtrl.TcDUT
TYPE ShortTestCtrl : 
STRUCT
	bStart :BOOL; //数据读取开始
	bDone  :BOOL; //数据读取完成
	Init:BOOL;//测试仪初始化开始
	InitFinish:BOOL;//测试仪初始化完成
   	iResult:INT; // 1 OK  2 NG
	
	ErrorID1 :BOOL;
	ErrorID2 :BOOL;

	Measure	:REAL;//电阻值
	Voltage	:REAL;//电压值
	TestTime:REAL;//测试时间
END_STRUCT
END_TYPE

// ---- P3UDTs/P3_ShortTest/ShortTestReceiveData.TcDUT
TYPE ShortTestReceiveData :
UNION
	sData 		: STRING(32);//CMD
	arrData 	 AT  %I*  :ARRAY [1..32] OF USINT;//ASCLL
END_UNION
END_TYPE

// ---- P3UDTs/P3_ShortTest/ShortTestSendData.TcDUT
TYPE ShortTestSendData :
UNION
	sData 		: STRING(32);//CMD
	arrData 	 AT  %Q*  :ARRAY [1..32] OF USINT;//ASCLL
END_UNION
END_TYPE

// ---- P3UDTs/P3_ShortTest/ST_ReceiveTestStatus.TcDUT
TYPE ST_ReceiveTestStatus :
STRUCT
	TransmitDone        :BOOL;   //数据发送完成
    ReceiveRequest      :BOOL;    
    InitAccepted        :BOOL;
    SndBufferFull       :BOOL;
    PutDataDone         :BOOL;
    InputLength         :USINT;
    TotalInputLength    :UINT;
END_STRUCT
END_TYPE

// ---- P3UDTs/P3_ShortTest/ST_SendTestStatus.TcDUT
TYPE ST_SendTestStatus :
STRUCT
	TransmitRequest          :BOOL;
	ReceiveAccepted          :BOOL;
	InitRequest              :BOOL;//
	PutData                  :BOOL:=TRUE;
	OutputLength             :UINT;//字节长度
END_STRUCT
END_TYPE

// ---- P3UDTs/P3_Temperature/STTempCtrl.TcDUT
TYPE STTempCtrl :
STRUCT
   In         AT  %I* :    TempIn;
   Out       AT  %Q* : TempOut;
   Tem_fPV :			  REAL; //当前温度
   fPVShow_1:			  REAL; //显示温度_1
   fPVShow1 :             REAL; //显示温度1
   fPVShow2 :             REAL; //显示温度2
   fPVShow3 :             REAL; //显示温度3
   fPVShow4 :             REAL; //显示温度4
   fPVShow5 :             REAL; //显示温度5
(***输出*)
 //  fTempMax                                :REAL;     //温度上限   监控
  // fTempMin                                 :REAL;     //温度下限   监控
(***Status*)
  bTempError_HI       :BOOL;     //超温报警
  bTempError_LI       :BOOL;     //超低温报警
  bSenserError         :BOOL;     //温度检测不一致
  bTuningError          :BOOL;     //自整定故障

END_STRUCT
END_TYPE

// ---- P3UDTs/P3_Temperature/ST_ParTemperature.TcDUT
TYPE ST_ParTemperature ://   温控相关参数
STRUCT
   fTempSet                                   	:REAL;// 设定温度温度(转换后)
   fTempOffset                              	:REAL;// 设定温度温度(转换后);// 温度偏移
	Tem_Offset									:REAL;//人工温度偏移
   fTempMax                                		:REAL;     //温度高限设置

  fTempArea                                     :REAL:=5;   //控制热电偶与监控热电偶温度偏差  

END_STRUCT
END_TYPE

// ---- P3UDTs/P3_Temperature/TempIn.TcDUT
TYPE TempIn :
STRUCT
     (****INPUT**)
   iPV:                                  INT;// 读取当前温度 (模块) 
   fPV:                                  REAL;// 读取当前温度(转换后)



  (****Status**)
   SaveParaOK:                      BOOL;           //保存参数OK
   PIDON:                             BOOL;          //PID功能开启
   AutoTuningON:                  BOOL;          //自整定开启
   AutoTuningerr:                   BOOL;          //自整定故障
   HeatingON:                       BOOL;          //加热中
   CoolingON:                       BOOL;          //制冷中
   AutoTuningOK:                  BOOL;          //自整定OK

END_STRUCT
END_TYPE

// ---- P3UDTs/P3_Temperature/TempInShow.TcDUT
TYPE TempInShow :  //最多5个备用通道
STRUCT
   iPV1:                                  INT:=9999;// 读取当前温度 (模块) 
   fPV1:                                  REAL;// 读取当前温度(转换后)

   iPV2:                                  INT:=9999;// 读取当前温度 (模块) 
   fPV2:                                  REAL;// 读取当前温度(转换后)

   iPV3:                                  INT:=9999;// 读取当前温度 (模块) 
   fPV3:                                  REAL;// 读取当前温度(转换后)

   iPV4:                                  INT:=9999;// 读取当前温度 (模块) 
   fPV4:                                  REAL;// 读取当前温度(转换后)

   iPV5:                                  INT:=9999;// 读取当前温度 (模块) 
   fPV5:                                  REAL;// 读取当前温度(转换后)
END_STRUCT
END_TYPE

// ---- P3UDTs/P3_Temperature/TempOut.TcDUT
TYPE TempOut :
STRUCT
     (****Output**)
   iSV:                                    INT;// 设定温度 (模块) 
   fSV:                                    REAL;// 设定温度温度(转换后)
   iPV_Offset:                          INT;// 温度偏移
    fPV_Offset:                         REAL;// 温度偏移
  (****Ctrl_World**)
   PIDRun:                              BOOL;           //PID运行中
   AutoTunning:                      BOOL;           //自动整定中
   SavePara:                           BOOL;          //保存参数
   HotRedun:                          BOOL;          //开启冗余功能
   BIP:                                   BOOL;          //

END_STRUCT
END_TYPE

// ---- P3UDTs/P3_Thickness/ST_Thickness.TcDUT
TYPE ST_Thickness :
STRUCT
T_start :BOOL;
T_finish :BOOL;
T_OK     :BOOL;	
T_NG     :BOOL;
END_STRUCT
END_TYPE

// ---- P3UDTs/P3_Torque/ST_TorqueMotion.TcDUT
TYPE ST_TorqueMotion :
STRUCT
	Velocity ,
	Acc,
	Dec,
	Jerk : REAL;
	
	FastReachVelo,
	BufferVelo 
	: REAL;
	
END_STRUCT
END_TYPE

// ---- P3UDTs/P3_Torque/ST_Torque_P3.TcDUT
TYPE ST_Torque_P3 :
STRUCT
	
	ColdpreLineTorSet:INT;//冷呀上料夹平移报警力矩设定
	ColdpreRetractTorSet:INT;//冷压上料夹进退报警力矩设定
	ColdpreWhirlTorSet:INT;//冷压上料夹旋转报警力矩设定
	ColdpreActTorSet:INT;//冷压驱动报警力矩设定
	OvenCarryTorSet:INT;//烤箱上料夹搬运报警力矩设定
	OvenRetractTorSet:INT;//烤箱上料夹进退报警力矩设定
	HotpreActTorSet:INT;//热压驱动报警力矩设定
	WeighLineTorSet:INT;//称重上料夹平移报警力矩设定
	WeighWhirlTorSet:INT;//称重上料夹旋转报警力矩设定
	SortingCarryTorSet:INT;//电芯分选夹搬运报警力矩设定
	OffloadCarryTorSet:INT;//电芯下料夹搬运报警力矩设定
	
	TapeAdvanceTorSet:INT;//后段贴胶平移实时力矩设定
	TapeTranslationTorSet:INT;//后段贴胶头进退实时力矩设定
	
	ColdpreLineTor:INT;//冷呀上料夹平移实时力矩
	ColdpreRetractTor:INT;//冷压上料夹进退实时力矩
	ColdpreWhirlTor:INT;//冷压上料夹旋转实时力矩
	ColdpreActTor:INT;//冷压驱动实时力矩
	OvenCarryTor:INT;//烤箱上料夹搬运实时力矩
	OvenRetractTor:INT;//烤箱上料夹进退实时力矩
	HotpreActTor:INT;//热压驱动实时力矩
	WeighLineTor:INT;//称重上料夹平移实时力矩
	WeighWhirlTor:INT;//称重上料夹旋转实时力矩
	SortingCarryTor:INT;//电芯分选夹搬运实时力矩
	OffloadCarryTor:INT;//电芯下料夹搬运实时力矩
	
	TapeAdvanceTor:INT;//后段贴胶平移实时力矩
	TapeTranslationTor:INT;//后段贴胶头进退实时力矩
	
	ColdpreLineTorAlarm:BOOL;//冷呀上料夹平移力矩超限报警
	ColdpreRetractTorAlarm:BOOL;//冷压上料夹进退力矩超限报警
	ColdpreWhirlTorAlarm:BOOL;//冷压上料夹旋转力矩超限报警
	ColdpreActTorAlarm:BOOL;//冷压驱动力矩超限报警
	OvenCarryTorAlarm:BOOL;//烤箱上料夹搬运力矩超限报警
	OvenRetractTorAlarm:BOOL;//烤箱上料夹进退力矩超限报警
	HotpreActTorAlarm:BOOL;//热压驱动力矩超限报警
	WeighLineTorAlarm:BOOL;//称重上料夹平移力矩超限报警
	WeighWhirlTorAlarm:BOOL;//称重上料夹旋转力矩超限报警
	SortingCarryTorAlarm:BOOL;//电芯分选夹搬运力矩超限报警
	OffloadCarryTorAlarm:BOOL;//电芯下料夹搬运力矩超限报警
	
	TapeAdvanceTorSetAlarm:BOOL;//后段贴胶平移实时力矩超限报警
	TapeTranslationTorSetAlarm:BOOL;//后段贴胶头进退实时力矩超限报警
	
	

END_STRUCT
END_TYPE

// ---- P3UDTs/P3_Variable/ST_StickIDGlue_date.TcDUT
TYPE ST_StickIDGlue_date :
STRUCT
StandbyCode_Step1			:UINT;//二维码拉胶自动步
StandbyCode_Step2			:UINT;//二维码取胶自动步	
PermitFilling				:BOOL;//允许上电芯信号
PermitMaterial				:BOOL;//允许下电芯信号
StandbyCode_Start			:BOOL;//备二维码胶开始信号
StandbyCode_Finish			:BOOL;//二维码取胶完成信号
StandbyCode_Done			:BOOL;//二维码胶拉胶完成信号

ScanCode_start				:BOOL;//扫码开始(流程)
ScanCode_AgainStart			:BOOL;//扫码复扫(流程)
ScanCode_finish				:BOOL;//扫码完成(流程)

StickGluePhoto_start   		:BOOL;//贴胶检测开始
StickGluePhoto_finish   	:BOOL;//贴胶检测完成

Code_State 					:INT;//扫码	1、OK,	2、NG
Code_State_1				:INT;//扫码	1、OK,	2、NG(切刀后结果)
Code_State_2				:INT;//扫码	1、OK,	2、NG(贴胶头结果）
Scan_IP						:STRING;//二维码扫码枪IP地址
bTcpOpen 					:BOOL;//扫码Tcp 连接
bScan_init 					:BOOL;//扫码初始化
bTcpOpen_OK 				:BOOL;//扫码Tcp 连接OK
bScan_start 				:BOOL;//扫码启动
//bCodeConError 				:BOOL;//扫码Tcp报错
//bCodeError  				:BOOL;//扫码故障
strCode   					:STRING;//电芯条码
strCode_1					:STRING;//电芯条码(切刀后记忆)
strCode_2					:STRING;//电芯条码(贴胶头记忆）
Scan_bDone 					:BOOL;//扫码完成	

IDGlueNumberOK    :BOOL;   //二维码胶料号OK

StickGluNgSet:INT;//外观检测NG连续计数设定值


END_STRUCT
END_TYPE

// ---- P3UDTs/P3_Weight/ST_Gross.TcDUT
TYPE ST_Gross :
STRUCT
	Weight_start :BOOL;//称重开始
	Weight_finish :BOOL;//称重完成
	Clear_start :BOOL;//清零开始
	Clear_finish :BOOL;//清零完成
	bweight	:REAL;
	Init	 :BOOL;//初始位
	error	:ARRAY[1..6] OF BOOL;
END_STRUCT
END_TYPE

// ---- P3UDTs/P3_Weight/ST_ReceiveData.TcDUT
TYPE ST_ReceiveData :
STRUCT
	  Status      AT  %I*     : ST_ReceiveStatus;   
      Data        AT  %I*     : ARRAY[0..31]OF USINT;
END_STRUCT
END_TYPE

// ---- P3UDTs/P3_Weight/ST_ReceiveStatus.TcDUT
TYPE ST_ReceiveStatus :
STRUCT
	TransmitDone        :BOOL;   //数据发送完成
    ReceiveRequest      :BOOL;    
    InitAccepted        :BOOL;
    SndBufferFull       :BOOL;
    PutDataDone         :BOOL;
    InputLength         :USINT;
    TotalInputLength    :USINT;
	
END_STRUCT
END_TYPE

// ---- P3UDTs/P3_Weight/ST_SendData.TcDUT
TYPE ST_SendData :
STRUCT
	  Status      AT  %Q*     : ST_SendStatus;   
      Data        AT  %Q*     : ARRAY[0..31]OF USINT;
END_STRUCT
END_TYPE

// ---- P3UDTs/P3_Weight/ST_SendStatus.TcDUT
TYPE ST_SendStatus :
STRUCT
	TransmitRequest          :BOOL;
	ReceiveAccepted          :BOOL;
	InitRequest              :BOOL;//
	PutData                  :BOOL:=TRUE;
	OutputLength             :UINT;//字节长度
	
	
	
	
END_STRUCT
END_TYPE

// ---- P2GVLs/GCylinder.TcGVL
	
VAR_GLOBAL
	arrCyCtrl			                  :ARRAY[1..MaxCy] OF ST_CyCtrl;	(*气缸控制接口*)
    AA1: INT;
END_VAR

VAR_GLOBAL CONSTANT

    MaxP2Cy                          	:UINT:=220;
	MaxCy			                  	:UINT:=295;		(*气缸数量*)
END_VAR

// ---- P2GVLs/GMotion.TcGVL
	
VAR_GLOBAL
	arrAxis			                      :ARRAY[1..MaxAxes] OF  axis_ref;		(*PTP轴*)
	arrAxisCtrl			                  :ARRAY[1..MaxAxes] OF ST_AxisCtrl;	(*轴的PTP控制接口*)

	
	arrDustMotor			              :ARRAY[1..Max_Dust] OF  ST_Dust_Motor;		(*毛刷电机*)
  	DrivesOP 		                       AT %I*		:ARRAY[1..155]OF UINT ;		                                 (*实际驱动器作为EtherCAT伺服的个数  ETHERCAT状态*)
	iActDriveMode	                   AT%I*	    	:ARRAY[1..3]OF SINT;			                                 (*驱动器返回的控制模式*)
    iSetDriveMode 	                  AT %Q*    	:ARRAY [1..3] OF SINT := [3(10)] ;          (*驱动器的模式输出，8为位置模式*)

	iMaxProfileVelo                   AT%Q* 	   :ARRAY[1..3]OF UDINT:=[3(139810133)];       (*单位为0.1rpm  500*2(23)   *)
	iPostiveTorqueLimits            AT%Q* 	  :ARRAY[1..3]OF UINT:=[3(2000)];
    iNegtiveTorqueLimits           AT%Q*     :ARRAY[1..3]OF UINT:=[3(2000)];
	iActTorque_D				AT%I*	    	:ARRAY[1..MaxAxes]OF INT;	//叠台后端轴力矩反馈值
	HMI_TorAlarm_D				:ARRAY[1..MaxAxes]OF BOOL ;	//叠台、后段各轴力矩过大报警(防止撞机)
END_VAR

VAR_GLOBAL CONSTANT
    MaxP2Axes		     	:UINT:=155;	
	MaxAxes				 	:UINT:=185;		(*轴数，不同于驱动器数，后者是物理轴的个数*)
    NumOfDrives			    :UINT:=185;		(*实际驱动器数*)
	iEcatOp			     	:UINT:=8;
	CSP					    :USINT:=8;
	CSV					    :USINT:=9;
	CST					    :USINT:=10;
	Max_Dust				:UINT:=3;
END_VAR

VAR_GLOBAL PERSISTENT
//VAR_GLOBAL
	iTargetTorque	                  AT%Q*    	:ARRAY[1..3]OF INT:= [3(-50)];			                     (*单位为0.1%*)
	arrAxisPar		   	:ARRAY[1..MaxAxes] OF ST_Axis_Par;	(*轴的PTP控制接口*)
	HMI_TorErrLimt_D			:ARRAY[1..MaxAxes]OF INT:=[MaxAxes(2000)]  ;//叠台、后段各轴力矩报警值设定
END_VAR



















	//aAxis_NcParam			:ARRAY[1..MaxAxes] OF ST_AxisParameterSet;	(*system manager中的NC参数读取*)
	//aReadNcParam			:ARRAY[1..MaxAxes] OF MC_ReadParameterSet; //FB
	//aWriteNcParam	        :ARRAY[1..MaxAxes] OF MC_WriteParameter;  //system manager中的NC参数写入
    //  mc_AxisParameter2       :E_AxisWritePar;




(************************************************************************************)
	(*欧姆龙驱动器力矩模式
	输出：
		6071 目标扭矩  INT16    0.1%  -5000~5000   （建议设置为PDO
		6072 最大扭矩 UINT16    0.1%  0~5000		（建议在驱动器中设置好
		3031 -01  力矩模式下的速度限制 单位rpm ，0-20000  INT32   出厂20000
	输入：当前力矩 6072
	*)
	(*
(*0821增加张力伺服参数*)
	iTartgetTorque	AT%Q*:ARRAY[2..2]OF INT:=[-80,80];		(*单位为0.1%*)
	iMaxVelo		AT%Q*:ARRAY[2..2]OF UDINT:=NumOfDancers[8000];	(*单位为0.1rpm*)
	iActualTorque	AT%I* :ARRAY[2..2]OF  INT;							(*单位为0.1%*)
	iSetDriveMode 	AT %Q*		:ARRAY [1..NumOfDrives] OF SINT := NumOfDrives[CSP];	(*驱动器的模式输出，8为位置模式*)
*)

// ---- P2GVLs/GVL_Par.TcGVL
VAR_GLOBAL    //参数
         parMachine            : ST_ParMachine;   //机械参数常量
         parTableNo          :  ST_ParTableNo;// 凸轮表号
END_VAR

VAR_GLOBAL PERSISTENT
	 //  parProduct                : ST_ParProduct;   //工艺参数
       parFilterAD              :ARRAY[1..MaxAINo] OF ST_ParFilterAD;
       parDA                     :ARRAY[1..44] OF INT;   //模拟量输出
	   DT_FingerprintKey:ST_FingerprintKey; //指纹解锁
	   
	   DT1_Timedata: FB_DTData;
	   DT2_Timedata:  FB_DTData;
	   DT3_Timedata:  FB_DTData;	   
END_VAR

VAR_GLOBAL PERSISTENT
//VAR_GLOBAL	
//	  iModeEN             : IModeEN;//功能屏蔽
	 	 P2M1_Par            : Parameters;
	 	 P2M2_Par            : Parameters;
	 	 P2M3_Par            : Parameters;
	 	 P2User1_Par        : User1_Par;
	  
	  	bDataValid:BOOL;//数据有效标志位
END_VAR

// ---- P2GVLs/GVL_User2.TcGVL
VAR_GLOBAL
(***P2M1*)
           stCarryingLineCam1_An                      :ST_Cam;
           stCarryingLineCam2_An                       :ST_Cam;
		   stCarryingLineCam3_An                      :ST_Cam;
           stCarryingLineCam4_An                       :ST_Cam;
		   stCarryingLineCam5_An                      :ST_Cam;
           stCarryingLineCam6_An                       :ST_Cam;		   
           sCarryingUpdown1_An                        :ST_Cam;
           sCarryingUpdown2_An                      :ST_Cam;
           sCarryingUpdown3_An                     :ST_Cam;
           sCarryingUpdown4_An                     :ST_Cam;

	       stCarryingLineCam1_Ca                    :ST_Cam;
           stCarryingLineCam2_Ca                      :ST_Cam;
		   stCarryingLineCam3_Ca                      :ST_Cam;
           stCarryingLineCam4_Ca                       :ST_Cam;	   
           sCarryingUpdown1_Ca                        :ST_Cam;
           sCarryingUpdown2_Ca                      :ST_Cam;
           sCarryingUpdown3_Ca                     :ST_Cam;
           sCarryingUpdown4_Ca                     :ST_Cam;	   
		   sPreneedleUpdown_Left   					:ST_Cam;	 
		   sPreneedleLine_Left   					:ST_Cam;	

		   sPreneedleUpdown_Right   					:ST_Cam;	 
		   sPreneedleLine_Right  					:ST_Cam;			   
		   
		   
		   sSEPTATLine1  						:ST_Cam;	
		   sSEPTATLine2							:ST_Cam;			   
		   
           stP2M1UnwindingTen                        :ST_Tension;








END_VAR

// ---- P2GVLs/GVL_User3.TcGVL

VAR_GLOBAL


(***方法***)
            stMethod                                 :ST_Method;

            bAllTenReady                              :BOOL;
            bAllGearReady                            :BOOL;
            bAllHomeReady                          :BOOL;


            bP1CamInReady                           :BOOL;
            bP2CamInReady_U                       :BOOL;
            bP2CamInReady_D                       :BOOL;
            bP3CamInReady_U                       :BOOL;
            bP3CamInReady_D                       :BOOL;

(***条件***)
           bAllTenOk                                   :BOOL;
           bHomeOk                                   :BOOL;        
           bAllGearOK                                :BOOL;
           bAllTempOK                               :BOOL;
           bAllRecOK                                  :BOOL;
           bAllCreatTableOK                        :BOOL;
           bAllCamOK                                 :BOOL;

(**报警**)
         arrCYOnAlarm                                :ARRAY[1..MaxCy]  OF BOOL;              //气缸ON报警
         arrCYOFFAlarm                              :ARRAY[1..MaxCy]  OF BOOL;              //气缸ON报警
         bCYHaveAlarm                              :BOOL;                                              //气缸有报警
		 P2M1_DTCYHaveAlarm                         :BOOL;                                              //一号叠台气缸有报警
		 P2M1_WJCYHaveAlarm                         :BOOL;                                              //一号尾卷贴胶气缸有报警

		 P2M2_DTCYHaveAlarm                         :BOOL;                                              //二号叠台气缸有报警
		 P2M2_WJCYHaveAlarm                         :BOOL;                                              //二号尾卷贴胶气缸有报警

		 P2M3_DTCYHaveAlarm                         :BOOL;                                              //三号叠台气缸有报警
		 P2M3_WJCYHaveAlarm                         :BOOL;                                              //三号尾卷贴胶气缸有报警

		 
         arrAxisbstop                                  :ARRAY[1..MaxAxes]  OF BOOL;            //轴停止
         arrAxisAlarm                                  :ARRAY[1..MaxAxes]  OF BOOL;            //轴报警
         bAxisHaveAlarm                              :BOOL;                                             //轴有报警
		 P2M1_DTAxisHaveAlarm                              :BOOL;                                             //一号叠台轴有报警
		 P2M1_WJAxisHaveAlarm                              :BOOL;                                             //一号尾卷轴有报警
		 
		 P2M1_AnHaveAlarm                              :BOOL;                                             //一号正极取料自动程序有报警
		 P2M1_CaHaveAlarm                              :BOOL;                                             //一号负极取料自动程序有报警
		 P2M1_DTHaveAlarm                              :BOOL;                                             //一号叠台自动程序有报警
		 P2M1_WJHaveAlarm                              :BOOL;                                             //一号尾卷自动程序有报警
		 P2M1_TJHaveAlarm                              :BOOL;                                             //一号贴胶自动程序有报警
		 P2M1_DoorAlarm                                :BOOL;                                             //一号叠台门禁报警
		 
		 P2M2_DTAxisHaveAlarm                              :BOOL;                                             //二号叠台轴有报警
		 P2M2_WJAxisHaveAlarm                              :BOOL;                                             //二号尾卷轴有报警

		 P2M2_AnHaveAlarm                              :BOOL;                                             //二号正极取料自动程序有报警
		 P2M2_CaHaveAlarm                              :BOOL;                                             //二号负极取料自动程序有报警
		 P2M2_DTHaveAlarm                              :BOOL;                                             //二号叠台自动程序有报警
		 P2M2_WJHaveAlarm                              :BOOL;                                             //二号尾卷自动程序有报警
		 P2M2_TJHaveAlarm                              :BOOL;                                             //二号贴胶自动程序有报警
		 P2M2_DoorAlarm                                :BOOL;                                             //二号叠台门禁报警
		 
		 P2M3_DTAxisHaveAlarm                              :BOOL;                                             //三号叠台轴有报警
		 P2M3_WJAxisHaveAlarm                              :BOOL;                                             //三号尾卷轴有报警		 
		 P2M3_AnHaveAlarm                              :BOOL;                                             //三号正极取料自动程序有报警
		 P2M3_CaHaveAlarm                              :BOOL;                                             //三号负极取料自动程序有报警
		 P2M3_DTHaveAlarm                              :BOOL;                                             //三号叠台自动程序有报警
		 P2M3_WJHaveAlarm                              :BOOL;                                             //三号尾卷自动程序有报警
		 P2M3_TJHaveAlarm                              :BOOL;                                             //三号贴胶自动程序有报警
		 P2M3_DoorAlarm                                :BOOL;                                             //三号叠台门禁报警
(*
         arrTemHIAlarm                              :ARRAY[1..MaxTemp]  OF BOOL;        //超温报警
         arrTemSenserAlarm                       :ARRAY[1..MaxTemp]  OF BOOL;        //温度检测不一致
         arrTemTuningAlarm                       :ARRAY[1..MaxTemp]  OF BOOL;        //自整定故障
         bTemHaveAlarm                            :BOOL;                                             //温控有报警
*)
          arrTenAlarm                                 :ARRAY[1..15]  OF BOOL;                  //张力报警
          bTenHaveAlarm                            :BOOL;                                           //张力有报警

          arrRecAlarm                                 :ARRAY[1..15]  OF BOOL;                  //纠偏报警
          bRecHaveAlarm                            :BOOL;                                          //纠偏有报警

         arrCreatTableAlarm                         :ARRAY[1..30]  OF BOOL;             //创建凸轮报警
         bCreatTableHaveAlarm                    :BOOL;//凸轮耦合有报警

         arrCamInAlarm                               :ARRAY[1..30]  OF BOOL;             //凸轮耦合报警
         bCamHaveAlarm                             :BOOL;//凸轮耦合有报警

         arrGearAlarm                                  :ARRAY[1..25]  OF BOOL;             //齿轮报警
         bGearHaveAlarm                             :BOOL;//凸轮耦合有报警


       fP1PutInPeacePos                                 :LREAL; //P1入片位置mm
       fP1PutInPeaceLength                             :REAL; //P1入片当前距离

       fP2PutInPeacePos                               :LREAL; //P1入片位置mm
       fP2PutInPeaceLength                          :REAL; //P1入片当前距离


        Axis_error                             :ARRAY[1..185]  OF BOOL;             //轴手自动对比报警

		P2M1_DError                                :BOOL;                                             //1号叠台门禁先报警
		P2M2_DError                                :BOOL;                                             //2号叠台门禁先报警
		P2M3_DError                                :BOOL;                                             //3号叠台门禁先报警


























END_VAR

// ---- P2GVLs/IO.TcGVL
VAR_GLOBAL

//////////////////////////叠片交互////////////////////////////////DP
AnMQ_MES1	                  AT %I*    	:ST_BeltData; //叠台1  MES交互
CaMQ_MES1	                  AT %I*    	:ST_BeltData; //叠台1  MES交互
AnMQ_MES2	                  AT %I*    	:ST_BeltData; //叠台2  MES交互
CaMQ_MES2	                  AT %I*    	:ST_BeltData; //叠台2 MES交互
AnMQ_MES3	                  AT %I*    	:ST_BeltData; //叠台3  MES交互
CaMQ_MES3	                  AT %I*    	:ST_BeltData; //叠台3  MES交互	

//预留数据交互
YL_I      		    AT %I*:ARRAY[1..50] OF BOOL ; //预留 1、气压不足报警；2、叠台一储气罐压力、3、叠台二储气罐压力、4、叠台三储气罐压力
YL_Q     				AT %Q*:ARRAY[1..50] OF BOOL ; //预留输；
YL_INT1     		AT %I*:ARRAY[1..50] OF INT  ; //预留输入INT；
YL_INT2     		AT %Q*:ARRAY[1..50] OF INT  ; //预留输出INT；
YL_GVL  :ARRAY [1..60] OF BOOL;//内部预留；1.叠台一正极送片流水线安全点动条件 2.叠台一负极送片流水线安全点动条件 3.叠台二正极送片流水线安全点动条件 4.叠台二负极送片流水线安全点动条件 5.叠台三正极送片流水线安全点动条件 6.叠台三负极送片流水线安全点动条件

//风机；
 dDrauFan                   :ARRAY[1..30] OF BOOL;   	// 风机  1、风机1开 ；2、风机2开；


//网络拓扑状态
Network1_OP AT %I*        :ARRAY [1..50] OF UINT;
Network2_OP AT %I*        :ARRAY [1..50] OF UINT;
Network3_OP AT %I*        :ARRAY [1..50] OF UINT;
Network4_OP AT %I*        :ARRAY [1..50] OF UINT;
Network5_OP AT %I*        :ARRAY [1..50] OF UINT;	

bNetwork1_OP  :ARRAY [1..50] OF BOOL;
bNetwork2_OP  :ARRAY [1..50] OF BOOL;
bNetwork3_OP  :ARRAY [1..50] OF BOOL;
bNetwork4_OP  :ARRAY [1..50] OF BOOL;
bNetwork5_OP :ARRAY [1..50] OF BOOL;	


//	与模切交互信号	
M_Pro    AT %I*: MToD_Process;//只读 模切生产过程信号
M_Sys    AT %I*: MToD_System;//只读 模切系统信号

D_Pro    AT %Q*: DToM_Process;//只写 叠片生产过程信号
D_Sys    AT %Q*: DToM_System;//只写 叠片系统信号

//P2M1 输入、输出信号
	I301 AT %I* :ARRAY [1..16] OF BOOL; //输入信号
	I302 AT %I* :ARRAY [1..16] OF BOOL; //输入信号
	I303 AT %I* :ARRAY [1..16] OF BOOL; //输入信号
	I304 AT %I* :ARRAY [1..16] OF BOOL; //输入信号
	I305 AT %I* :ARRAY [1..16] OF BOOL; //输入信号
	I306 AT %I* :ARRAY [1..16] OF BOOL; //输入信号
	I307 AT %I* :ARRAY [1..16] OF BOOL; //输入信号
	I308 AT %I* :ARRAY [1..16] OF BOOL; //输入信号	
	I309 AT %I* :ARRAY [1..16] OF BOOL; //输入信号	
	
	Q301 AT %Q* :ARRAY[1..16] OF BOOL;//输出信号
	Q302 AT %Q* :ARRAY[1..16] OF BOOL;//输出信号
	Q303 AT %Q* :ARRAY[1..16] OF BOOL;//输出信号
	Q304 AT %Q* :ARRAY[1..16] OF BOOL;//输出信号
	Q305 AT %Q* :ARRAY[1..16] OF BOOL;//输出信号
	Q306 AT %Q* :ARRAY[1..16] OF BOOL;//输出信号
	Q307 AT %Q* :ARRAY[1..16] OF BOOL;//输出信号
	Q308 AT %Q* :ARRAY[1..16] OF BOOL;//输出信号
	Q309 AT %Q* :ARRAY[1..16] OF BOOL;//输出信号
	
	
	
	AI30 AT %I* :ARRAY [1..9] OF INT; //模拟量输入信号
	AO30 AT %Q* :ARRAY [1..9] OF INT; //模拟量输出信号


//P2M2 输入、输出信号
	I401 AT %I* :ARRAY [1..16] OF BOOL; //输入信号
	I402 AT %I* :ARRAY [1..16] OF BOOL; //输入信号
	I403 AT %I* :ARRAY [1..16] OF BOOL; //输入信号
	I404 AT %I* :ARRAY [1..16] OF BOOL; //输入信号
	I405 AT %I* :ARRAY [1..16] OF BOOL; //输入信号
	I406 AT %I* :ARRAY [1..16] OF BOOL; //输入信号
	I407 AT %I* :ARRAY [1..16] OF BOOL; //输入信号
	I408 AT %I* :ARRAY [1..16] OF BOOL; //输入信号
	I409 AT %I* :ARRAY [1..16] OF BOOL; //输入信号
	
	Q401 AT %Q* :ARRAY[1..16] OF BOOL;//输出信号
	Q402 AT %Q* :ARRAY[1..16] OF BOOL;//输出信号
	Q403 AT %Q* :ARRAY[1..16] OF BOOL;//输出信号
	Q404 AT %Q* :ARRAY[1..16] OF BOOL;//输出信号
	Q405 AT %Q* :ARRAY[1..16] OF BOOL;//输出信号
	Q406 AT %Q* :ARRAY[1..16] OF BOOL;//输出信号
	Q407 AT %Q* :ARRAY[1..16] OF BOOL;//输出信号
	Q408 AT %Q* :ARRAY[1..16] OF BOOL;//输出信号
	Q409 AT %Q* :ARRAY[1..16] OF BOOL;//输出信号
	
	AI40 AT %I* :ARRAY [1..9] OF INT; //模拟量输入信号
	AO40 AT %Q* :ARRAY [1..9] OF INT; //模拟量输出信号	
	
//P2M3 输入、输出信号
	I501 AT %I* :ARRAY [1..16] OF BOOL; //输入信号
	I502 AT %I* :ARRAY [1..16] OF BOOL; //输入信号
	I503 AT %I* :ARRAY [1..16] OF BOOL; //输入信号
	I504 AT %I* :ARRAY [1..16] OF BOOL; //输入信号
	I505 AT %I* :ARRAY [1..16] OF BOOL; //输入信号
	I506 AT %I* :ARRAY [1..16] OF BOOL; //输入信号
	I507 AT %I* :ARRAY [1..16] OF BOOL; //输入信号
	I508 AT %I* :ARRAY [1..16] OF BOOL; //输入信号
	I509 AT %I* :ARRAY [1..16] OF BOOL; //输入信号
	
	Q501 AT %Q* :ARRAY[1..16] OF BOOL;//输出信号
	Q502 AT %Q* :ARRAY[1..16] OF BOOL;//输出信号
	Q503 AT %Q* :ARRAY[1..16] OF BOOL;//输出信号
	Q504 AT %Q* :ARRAY[1..16] OF BOOL;//输出信号
	Q505 AT %Q* :ARRAY[1..16] OF BOOL;//输出信号
	Q506 AT %Q* :ARRAY[1..16] OF BOOL;//输出信号
	Q507 AT %Q* :ARRAY[1..16] OF BOOL;//输出信号
	Q508 AT %Q* :ARRAY[1..16] OF BOOL;//输出信号
	Q509 AT %Q* :ARRAY[1..16] OF BOOL;//输出信号
	
	AI50 AT %I* :ARRAY [1..9] OF INT; //模拟量输入信号
	AO50 AT %Q* :ARRAY [1..9] OF INT; //模拟量输出信号	
//P2传感器信号、按钮
	P2Senser :ST_P2Senser;//传感器信号
	P2Btn    :ST_P2Button;//按钮
END_VAR

VAR_GLOBAL CONSTANT
	MaxAINo				:INT:=52;		(*ai通道数量*)
END_VAR

// ---- P2GVLs/N.TcGVL

VAR_GLOBAL  //常量
(**轴**)  
	P2AxisNo:      ST_P2AxisName;
    VirAxisNo:      ST_P2VirAxisName;
(**气缸**)
	P2CYNo:        ST_P2CylinderName;
(**电磁阀**)
	P2EVNo:        ST_P2ElectValveName;

(***纠偏**)
     RecNo:         ST_RecName;

(***温控*)
  //  TempNo:      ST_TempName;

(******凸轮表****)
    P2TableNo:      ST_TableName;

	//毛刷
	DustNo        :ST_Dust;

END_VAR

// ---- P2GVLs/System.TcGVL

VAR_GLOBAL	
	stHmiSysCmd			    	    :ST_SysCmd;
	MachimeVersion				:STRING:='V2024.5.28';(*当前系统版本号*)
	MachimeTpye					:STRING:='YKRFH';
	SysInfo						       :SystemInfoCtrl;
	fPlcCycleTime_ms			    :LREAL;
	pulse						            :PulseCtrl;	
	stTime: TIMESTRUCT;
    versionwrite  : BOOL;//版本号写入






END_VAR

// ---- P2GVLs/User01.TcGVL

VAR_GLOBAL
    stSysState :ST_SystemRUN;//系统状态机
	P2M1_DTSysState :ST_SystemRUN;//一号叠台系统状态机
	P2M1_WJSysState :ST_SystemRUN;//一号尾卷系统状态机
	
	
	 P2M2_DTSysState :ST_SystemRUN;//二号叠台系统状态机
	  P2M2_WJSysState :ST_SystemRUN;//二号叠台系统状态机
	 
	 P2M3_DTSysState :ST_SystemRUN;//三号叠台系统状态机
	 P2M3_WJSysState :ST_SystemRUN;//三号叠台系统状态机
	 
      arrda1:                         UINTARR2;
      fbPulseCtrl                  :ARRAY[1..10]   OF      PulseGeneratorCtrl;
	  Machine_No        :STRING;//机台编号
	 //系统信号
	P2_sysControl: System_Control;
	//1号叠片
	P2M1_program: P2Program_FB;
	P2M1_MachCtrl: ControlSignal;
	P2M1_sysControl: System_Control;
	P2M1_CycNo: EleControlNo;
	P2M1_Axise: P2_AxiseNo;
    P2M1_TableNo  : P2_TableNo;
	P2M1_CCD:ST_CCDCom;
	P2M1_Torque:ST_Torque;
	//2号叠片
	P2M2_program: P2Program_FB;
	P2M2_MachCtrl: ControlSignal;
	P2M2_sysControl: System_Control;
	P2M2_CycNo: EleControlNo;
	P2M2_Axise: P2_AxiseNo;
     P2M2_TableNo  : P2_TableNo;
	P2M2_CCD:ST_CCDCom;
	P2M2_Torque:ST_Torque;
	//3号叠片
	P2M3_program: P2Program_FB;
	P2M3_MachCtrl: ControlSignal;
	P2M3_sysControl: System_Control;
	P2M3_CycNo: EleControlNo;
	P2M3_Axise: P2_AxiseNo;	
    P2M3_TableNo  : P2_TableNo;
	P2M3_CCD:ST_CCDCom;
	P2M3_Torque:ST_Torque;
	

	bDiffVel:ARRAY [1..3] OF BOOL;//叠片速度不同标志位
END_VAR



































	(* 
  
   	 scRecipe :            CS_Recipe;
	 iRecipe:               IRecipe;
	 arriVirSingle:    ARRAY  [1..30] OF INT:=[30(1)] ;  //虚拟仿真信号
	 arriVirSingle2:  ARRAY [1..30] OF INT:=[30(1)] ;  //虚拟仿真信号
	 arriVirSingle3:  ARRAY [1..30] OF INT:=[30(1)] ;  //虚拟仿真信号


	arrAxisError :                ARRAY[1..MaxAxes] OF BOOL;//轴报警
	arrActuatorsError :        ARRAY[1..20] OF BOOL;//气缸
	arrFunctionError :         ARRAY[1..20] OF BOOL;//功能


	 cmd: CMD;
	 ShortDataShow:ShortDataShow; 
	 csShortTest :CS_ShortTest;
	 csCodeTcp: CS_CodeTcp;
	 IShort:IShortTest;
	 iCode:ICode;
	csCcdTcp:CS_CcdTcp_V2;
	iCCD:ICCD;
	ccdData:STCcdData;
	*)

// ---- P3GVLs/P3IO.TcGVL

VAR_GLOBAL
	
//P3 输入、输出信号
    I601 AT %I* :ARRAY [1..16] OF BOOL; //输入信号
	I602 AT %I* :ARRAY [1..16] OF BOOL; //输入信号
	I603 AT %I* :ARRAY [1..16] OF BOOL; //输入信号
	I604 AT %I* :ARRAY [1..16] OF BOOL; //输入信号
	I605 AT %I* :ARRAY [1..16] OF BOOL; //输入信号
	I606 AT %I* :ARRAY [1..16] OF BOOL; //输入信号
	I607 AT %I* :ARRAY [1..16] OF BOOL; //输入信号
	I608 AT %I* :ARRAY [1..16] OF BOOL; //输入信号
	I609 AT %I* :ARRAY [1..16] OF BOOL; //输入信号
	I701 AT %I* :ARRAY [1..16] OF BOOL; //输入信号
	I702 AT %I* :ARRAY [1..16] OF BOOL; //输入信号
	I703 AT %I* :ARRAY [1..16] OF BOOL; //输入信号
	
	Q601 AT %Q* :ARRAY [1..16] OF BOOL; //输出信号
	Q602 AT %Q* :ARRAY [1..16] OF BOOL; //输出信号
	Q603 AT %Q* :ARRAY [1..16] OF BOOL; //输出信号
	Q604 AT %Q* :ARRAY [1..16] OF BOOL; //输出信号
	Q605 AT %Q* :ARRAY [1..16] OF BOOL; //输出信号
	Q606 AT %Q* :ARRAY [1..16] OF BOOL; //输出信号
	Q607 AT %Q* :ARRAY [1..16] OF BOOL; //输出信号
	Q608 AT %Q* :ARRAY [1..16] OF BOOL; //输出信号
	Q609 AT %Q* :ARRAY [1..16] OF BOOL; //输出信号
	Q701 AT %Q* :ARRAY [1..16] OF BOOL; //输出信号
	Q702 AT %Q* :ARRAY [1..16] OF BOOL; //输出信号
	AI60 AT %I* :ARRAY [0..3] OF INT; //模拟量输入信号
	AO60 AT %Q* :ARRAY [0..3] OF INT; //模拟量输出信号	
	chengzhong		AT %I*  : 	USINT;//称重临时用
	ThicknessPar	AT %I*	:	DINT;//测厚参数(转化前)
	
	MTD_Mes1	AT%I* :MTD_Mes1;	//接收模切优报表数据XFP20240318
	DTM_Mes1	AT%Q* :DTM_Mes1;	//发送叠台信号至模切XFP20240318

    P3Senser :ST_P3Senser;//传感器信号
	P3Button :ST_P3Button;//按钮
	
	
	
	P3WeightRec:     ST_ReceiveData;  //
	P3WeightSend:    ST_SendData;  //
	

	P3ShortTestRec: 	ShortTestReceiveData;  //短路测试返回数据
	P3ShortTestSend  : 	ShortTestSendData;  //短路测试发送数据
	
	P3ShortSendCrtl AT  %Q*:    ST_SendTestStatus;//发送控制字
	P3ShortReCrtl   AT  %I*: 	ST_ReceiveTestStatus;//接收控制字
	
	Pass1:BOOL;//强制下料到1#；
	Pass2:BOOL;//强制下料到2#；
	
	Mes1	:Mes1;	//XFP20240315
END_VAR

// ---- P3GVLs/P3Motion.TcGVL

VAR_GLOBAL
	stP3NgPushMoter                       :ARRAY[1..4] OF ST_SetpMotor;


   	arrAxisCtrlV2                         :ARRAY[166..168] OF ST_AxisCtrlV2;


	ADSRefMark:BOOL;//ADS写入标志
	fADSWrite_Limit:ARRAY[1..12]OF ADSWrite_Limit;
	HMI_SetButton:ARRAY[1..12]OF  BOOL;//ADS软限位值写入
	HMI_ADSAlarm:ARRAY[1..12]OF  BOOL;//ADS软限位写入失败报警
	HMI_SaveBias:ARRAY[1..12] OF LREAL;//软限位读出数据
END_VAR



VAR_GLOBAL PERSISTENT
	
	arrAxisParV2        :ARRAY[166..168] OF ST_Axis_parV2;
	//	fSavePositionBias:ARRAY[1..4] OF LREAL;(*写入软限位的值*)
	//HMI_Button:ARRAY[1..4]OF  BOOL;//ADS软限位开关
END_VAR
VAR_GLOBAL CONSTANT
    MaxP3Axes		    :UINT:=185;	

END_VAR

// ---- P3GVLs/P3Name.TcGVL

VAR_GLOBAL  //常量
(**轴**)  
	P3AxisNo:      ST_P3AxisName;
(**气缸**)
	P3CYNo:        ST_P3CylinderName;
(**电磁阀**)

(***温控*)
    TempNo:      ST_TempName;
END_VAR

// ---- P3GVLs/P3Par.TcGVL

VAR_GLOBAL
	CellNo: ST_MemoryName;//电芯记忆编号
	Torque_P3:ST_Torque_P3;
END_VAR



VAR_GLOBAL PERSISTENT
  	P3User2_Par:              User2_Par;
	P3_Production:LocalProduction;//产能统计
	CellMemory: ARRAY [1..80] OF ST_CellMemory;// 电芯记忆
	P3Par :P3_Par;
	P3_Weight_gross	:ST_Gross;
	Alarm_CS :ARRAY[0..23] OF UDINT;//报警时间计数
	Auto_CS :ARRAY[0..23] OF UDINT;//运行时间计数
	Manul_CS :ARRAY[0..23] OF UDINT;//待机时间计数
	Oven_par :ARRAY[1..2] OF REAL;//烤箱升降取放烤箱辅助位(相对位置)
	P3TimeData :               FB_HDData;
	P3_PLC_PC_MES:ST_PLC_PC_MES;//PLC与PC物料码交互
	
	//模切、叠台条码交互
	DT_To_MQ_MES AT %Q*:ST_DT_To_MQ_MES;
	MQ_To_DT_MES AT %I*:ST_MQ_To_DT_MES;

END_VAR

// ---- P3GVLs/P3Press.TcGVL

VAR_GLOBAL
	
//	bStickStart:BOOL;//贴胶允许
//	bStickFinish:BOOL;//贴胶完成

	P3_Oven: ARRAY[1..21] OF INT;//烤箱名称映射	
	Oven_full: BOOL;//烤箱满电芯信号
	Oven_empty :BOOL;//烤箱全空信号
	Permit_Cold_Press   :BOOL;//允许冷压信号
	Permit_Hot_Press    :BOOL;//允许热压信号
	Permit_Weigh        :BOOL;//允许称重信号
	Permit_Thickness    :BOOL;//允许测厚信号
	
    Cold_Press_Finish   :BOOL;//冷压完成信号
	Hot_Press_Finish   :BOOL;//热压完成信号
	Weigh_Finish        :BOOL;//称重完成信号
	Thickness_Finish     :BOOL;//测厚完成信号
	ShortTest_Finish     :BOOL;//短路测试
    Coldbusy  :BOOL;//冷压z中
	Hotbusy  :BOOL;//热压中
	
	PermitColdPressRack :BOOL;//冷压允许上料信号
	PermitHotPressRack  :BOOL;//热压允许上料信号
	Permit_WeighRack     :BOOL;//允许称重上料信号
	Permit_ThicknessRack :BOOL;//允许测厚上料信号
	Permit_BlankingRack  :BOOL;//允许放料信号
	Permit_TakeMaterial  :BOOL;//允许取料
	Permit_ShortTest     :BOOL;//允许短路测试
	Permit_Blow:ARRAY[1..2] OF BOOL;//允许冷热压吹气，1：冷压，2：热压
	
	
	
	GlueFinish          :ARRAY[1..3] OF BOOL;//贴胶完成可下料信号
	Press_Clear         :ARRAY[1..2] OF BOOL;//1、冷压清零  2、热压清零
	Step30 :UINT;//贴胶下料流程
	Step31 :UINT;//冷压流程
	Step32 :UINT;//烤箱上下料流程
	Step33 :UINT;//热压流程
	Step34 :UINT;//称重上料流程
	Step35 :UINT;//分选流程
	Step36 :UINT;//下料流程
	Step37 :UINT;//备胶流程
	Step38 :UINT;//贴胶流程
	Step39 :UINT;//贴二维码胶流程
	TestOne:BOOL;//手动放料进冷压确定
	
	weight_step :UINT;//称重流程
	Step_Short :UINT;//短路测试
	P3_Press_PV: ARRAY [1..2] OF REAL;// 当前压力值
	P3_Torque_Act: ARRAY [1..2] OF REAL;// 扭矩当前值
	P3_T_achieve :ARRAY[1..42] OF BOOL;//烤箱温度达到信号
	P3_Hot_press :BOOL;//热压温度达到
	b_Alarm         :ARRAY[1..19] OF BOOL;//1、叠台1报警  2、叠台2报警  3、叠台3报警  4、尾段报警
	Alarm_bReset    :BOOL;//报警复位
	P3_SystemRUN    :ST_SystemRUN;//尾段系统
	LateBlanking_init_start :ARRAY[0..10] OF BOOL;//初始位开始,0、后段初始化 1、冷压上料初始化 2、冷压初始化 3、烤箱上下料初始化 4、热压初始化 5、称重上料初始化 6、分选初始化 7、下料初始化
	LateBlanking_init_OK 	:ARRAY[0..10] OF BOOL;//初始位完成,0、后段初始化 1、冷压上料初始化 2、冷压初始化 3、烤箱上下料初始化 4、热压初始化 5、称重上料初始化 6、分选初始化 7、下料初始化
	SingleStep           :ARRAY[1..10] OF BOOL;//单步
	StepModel            :ARRAY[1..10] OF BOOL;//单步模式 ON:单步中 OFF:连动中
	//Oven_cell_Shield     :ARRAY[1..42] OF BOOL;//烤箱电芯屏蔽
	//Oven_Shield          :ARRAY[1..21] OF BOOL;//烤箱屏蔽
	P3_Oven_Button          :ARRAY[1..42] OF BOOL;//烤箱位置一键按钮 
	P3_Oven_Flow            :ARRAY[1..42] OF BOOL;//烤箱位置到位显示 
	P3_Start                    :ARRAY[1..10] OF BOOL;//启动按钮
	ColdPress_start              :BOOL;//冷压开始
	HotPress_start              :BOOL;//热压开始
	b_Thickness                 :ST_Thickness;//测厚信号
	Thickness_Step  			:UINT;
	HD_Error           :ARRAY[1..99] OF BOOL; //后段其它报警
	b_Press_condition  :ARRAY[1..2] OF BOOL;//下压安全条件
	WeighLine_1 :REAL;//称重安全位置1
	WeighLine_2  :REAL;//称重安全位置2
	OvenCarrying_1 :REAL;//烤箱搬运安全位
	Sort_1         :REAL;//分选安全位1
	Sort_2         :REAL;//分选安全位2
	Offloading_1    :REAL;//下料平移安全位置
	Push_NG         :ARRAY[1..4] OF BOOL;//踢NG中信号
	Thickness_Par_Z		:REAL;//测厚参数(转化后)
	P3_Weight_clear	:ST_Gross;
	Pressing       : ARRAY[1..2] OF BOOL;//压力压合中
	P3_Error		:ARRAY[1..200] OF BOOL;//后段报警
	P3_Tem_Error    :ARRAY[1..96] OF BOOL;//温度未在范围内
	Tem_HOT			:BOOL;//一键加热
	Tem_Cold		:BOOL;//一键关闭加热
	T_Residue:   ARRAY[1..42] OF UDINT;
	Door_error : ARRAY[1..40] OF BOOL;//后段门禁报警
	bTcpOpen :BOOL;//扫码Tcp 连接
	bScan_init :BOOL;//扫码初始化
	bTcpOpen_OK :BOOL;//扫码Tcp 连接OK
	bScan_start :BOOL;//扫码启动
	bCodeConError :BOOL;//扫码Tcp报错
	bCodeError  :BOOL;//扫码故障
	strCode   :STRING;//冷压上料扫码码条
	Code_State :INT;//1、OK,2、NG
	Scan_bDone :BOOL;//扫码完成
	Scan_start	:BOOL;//扫码开始--扫码枪
	Scan_finish	:BOOL;//扫码完成--扫码枪
	
	FSY_An_bTcpOpen :BOOL;//负极风速仪Tcp 连接
	FSY_An_bScan_init :BOOL;//负极风速仪初始化
	FSY_An_bTcpOpen_OK :BOOL;//负极风速仪Tcp 连接OK
	FSY_An_bScan_start :BOOL;//负极风速仪读取启动
	FSY_An_bCodeConError :BOOL;//负极风速仪Tcp报错
	FSY_An_bCodeError  :BOOL;//负极风速仪故障
	FSY_An_Scan_bDone :BOOL;//负极风速仪读取完成
	FSY_An_Scan_start	:BOOL;//负极风速仪读取开始--风速仪
	FSY_An_Scan_finish:BOOL;//负极风速仪读取完成--风速仪

	FSY_Ca_bTcpOpen :BOOL;//正极风速仪Tcp 连接
	FSY_Ca_bScan_init :BOOL;//正极风速仪初始化
	FSY_Ca_bTcpOpen_OK :BOOL;//正极风速仪Tcp 连接OK
	FSY_Ca_bScan_start :BOOL;//正极风速仪读取启动
	FSY_Ca_bCodeConError :BOOL;//正极风速仪Tcp报错
	FSY_Ca_bCodeError  :BOOL;//正极风速仪故障
	FSY_Ca_Scan_bDone :BOOL;//正极风速仪读取完成
	FSY_Ca_Scan_start	:BOOL;//正极风速仪读取开始--风速仪
	FSY_Ca_Scan_finish:BOOL;//正极风速仪读取完成--风速仪
	
	IDStickStart:BOOL;//二维码贴胶开始
	IDStickFinish:BOOL;//二维码贴胶完成
	StickIDGlue			:ST_StickIDGlue_date;//二维码平台信号
	
	SHORT_HOT :ShortTestCtrl;//短路测试的控制
	
	Pressure_Alarm  : ARRAY[1..2] OF BOOL;//1.冷压压力报警  2.热压压力报警
	PC_start :BOOL;//上位机上传数据开始
	PC_finish :BOOL;//上位机上传数据完成
	PC_heart :BOOL;//上位机心跳
	PLC_heart :BOOL;//PLC心跳
	P3_manual :BOOL;//后段手动状态（用于HMI）
	Init_step :ARRAY[1..10] OF UINT;//初始化步
	Sampling_finish :ARRAY [1..2] OF BOOL;//采集完成
	Sampling_mean :ARRAY[1..2] OF REAL;//采集平均值
	PC_start1 :BOOL;//上位机上传数据开始1
	PC_finish1 :BOOL;//上位机上传数据完成1
	Cold_start :BOOL;//上位机判断开始
	Cold_finish :BOOL;//上位机判断完成
	Puttime :STRING;//投入时间
	Outtime :STRING;//产出时间
	PC_alarm :ARRAY[1..18] OF BOOL;//物料信息 1、正极膜卷用完，请更换物料号 2、负极膜卷用完，请更换物料号 3、蓝胶已经用完，请更换物料号 4、二维码胶已经用完，请更换物料号 5、隔膜1已经用完 6、隔膜2已经用完 7、隔膜3已经用完
	
	
	HMI_Year	:INT;//触摸屏时间（年）
	HMI_Month 	:INT;//触摸屏时间（月）
	HMI_day  	:INT;//触摸屏时间（日）
	HMI_Hour 	:INT ;//触摸屏时间（时）
	HMI_Minute 	:INT ;//触摸屏时间（分）
	HMI_Second 	:INT ;//触摸屏时间（秒）
	
	Day_Output :UINT;//白班总产量
	Night_Output :UINT;//夜班总产量
	Output_step :UINT;//产量统计
	Time_Output :ARRAY[0..23] OF UINT;//时段产量
	Day_Output_OK :UINT;//白班良品数
	Day_Output_NG :UINT;//白班不良品数
	Night_Output_OK :UINT;//夜班良品数
	Night_Output_NG :UINT;//夜班不良品数
	Day_Clear		:BOOL;//白班数量清零
	Night_Clear		:BOOL;//夜班数量清零
	Push_NG_condition :ARRAY[1..4] OF BOOL;//放NG料安全条件,1、放对齐度NG料安全条件,2、放短路NG料盒安全条件 3、放测厚NG料盒安全条件 4、放扫码NG或者MES的NG料盒安全条件
	Push_NG_Full :ARRAY[1..4] OF BOOL;//NG料盒满料信号 1、对齐度 2、短路 3、测厚 4、扫码或者MES
	PC_Error :BOOL;//上位机读取数据异常
	Day_NG    :Statistics;//白班NG分类
	Night_NG  :Statistics;//夜班NG分类
	Day_Yield   :REAL;//白班良率
	Night_Yield :REAL;//夜班良率
	Cold_Scan_code :BOOL;//冷压扫码复扫
	Oven_CYOFF_condition :BOOL;//烤箱已经全部关闭条件
	Oven_CYON_condition  :BOOL;//烤箱已经全部打开条件
	Oven_CY_STOP :BOOL;//烤箱气缸报警烤箱轴急停
	QY_error :BOOL;//总气压报警
	Oven_POS1 :BOOL;//烤箱进退初始位
	tip_1     :ARRAY[1..50] OF BOOL;//冷压上料提示
	tip_2     :ARRAY[1..50] OF BOOL;//冷压提示
	tip_3     :ARRAY[1..50] OF BOOL;//烤箱上下料提示
	tip_4     :ARRAY[1..50] OF BOOL;//热压提示
	tip_5     :ARRAY[1..50] OF BOOL;//称重上料提示
	tip_6     :ARRAY[1..50] OF BOOL;//1分选单步中 2.电芯NG1料盒锁定气缸未锁定 3.电芯NG2料盒锁定气缸未锁定 4.电芯NG3料盒锁定气缸未锁定
	tip_7     :ARRAY[1..50] OF BOOL;//下料提示
	tip_8     :ARRAY[1..30] OF BOOL;//烤箱上料时，对应烤箱门未打开
	tip_9     :ARRAY[1..30] OF BOOL;//烤箱下料时，对应烤箱门未打开
	tip_10     :ARRAY[1..21] OF BOOL;//烤箱上下料时，有门未关闭
	
	Oven_PB_condition :BOOL;//烤箱屏蔽条件
	fDataMax  :UDINT;//
	
	Make_sure : BOOL ;//确认
    Bullet_window : BOOL ;//弹窗触发
    Device_Status_code :INT ;//设备状态代码
    Manual_click_code  :INT ;//手动点选代码 
    Equipment_parameter_check :INT ;//设备参数校对
	
	ColdpreLineTorMark:BOOL;//冷呀上料夹平移力矩超限报警标志
	ColdpreRetractTorMark:BOOL;//冷压上料夹进退力矩超限报警标志
	ColdpreWhirlTorMark:BOOL;//冷压上料夹旋转力矩超限报警标志
	ColdpreActTorMark:BOOL;//冷压驱动力矩超限报警标志
	OvenCarryTorMark:BOOL;//烤箱上料夹搬运力矩超限报警标志
	OvenRetractTorMark:BOOL;//烤箱上料夹进退力矩超限报警标志
	HotpreActTorMark:BOOL;//热压驱动力矩超限报警标志
	WeighLineTorMark:BOOL;//称重上料夹平移力矩超限报警标志
	WeighWhirlTorMark:BOOL;//称重上料夹旋转力矩超限报警标志
	SortingCarryTorMark:BOOL;//电芯分选夹搬运力矩超限报警标志
	OffloadCarryTorMark:BOOL;//电芯下料夹搬运报警力矩设定
	
	StickerStandbyDone : BOOL;//备胶完成
	stickGlueDone : BOOL;//贴胶完成
	Uppercorepermit : BOOL;//放电芯允许
	Bottomsignal : BOOL;//贴胶下料信号
	StickerDoneNo1:ARRAY[0..9] OF BOOL;//已贴胶的道数
	Gluebtn	:BOOL;		//		拉胶按钮
	Cutbtn	:BOOL;		//		切胶按钮
	Readybtn	:BOOL;		//		备胶按钮
	
	HDQuery:BOOL;//时间查询
	HDdate:INT;//查询日期
	OEE:REAL;//稼动率	
	MQstate:INT;//模切状态   1:自动中   2:自动-Ready  3:手动   4:急停    5：报警    6.自动-NoReady
	OEE1:                             FB_OEE;//稼动率
	
	 P2SaveParDone      :BOOL;
	 P2ReadParDone     :BOOL;
	 
	 BlueGlueNumberOK:BOOL;//蓝胶条码校验OK
END_VAR

// ---- P3GVLs/P3Temperature.TcGVL

VAR_GLOBAL
   
    
   

END_VAR


VAR_GLOBAL PERSISTENT
	TempPVs                          AT %I* :  ARRAY[1..MaxTemp]  OF  TempInShow;//显示温控输入
	arrTempCtrl                         : ARRAY[1..MaxTemp]  OF  STTempCtrl;
	arrTempPar		                	:ARRAY[1..MaxTemp] OF   ST_ParTemperature;	(*轴的PTP控制接口*)
END_VAR

VAR_GLOBAL CONSTANT
	  MaxTemp			             	:UINT:=104;		(**温控数量*)
END_VAR

// ---- P2POUs/POUS/P2M1_Auto.TcPOU
PROGRAM P2M1_Auto






VAR
	DT1Code_MES: ARRAY[1..10] OF R_TRIG;
END_VAR

// 1号叠台自动
P2M1_program(
	DTselect:=1 , 
	Sys_Control:=P2M1_sysControl , 
	Mach_Control:=P2M1_MachCtrl , 
	arrCyNo:=P2M1_CycNo , 
	AxiseNo:=P2M1_Axise , 
	TableNo:=P2M1_TableNo,
	Par:=P2M1_Par ,
	CCD:=P2M1_CCD,
	Torque:=P2M1_Torque,
	iTargetTorqueTest=>iTargetTorque[1]
	);

//叠片给模切的信号
D_Pro.bAn_M1Done:=P2M1_MachCtrl.An_b.AN_BeltDone; //正极取流水线极片完成
D_Pro.bAn_M1Safety:=P2M1_MachCtrl.An_b.AN_BeltSafe;//正极取流水线安全位
D_Pro.bCa_M1Done:=P2M1_MachCtrl.Ca_b.Ca_BeltDone;//负极取水线极片完成
D_Pro.bCa_M1Safety:=P2M1_MachCtrl.Ca_b.Ca_BeltSafe;//负极取流水线安全位
//D_Sys.fM1MainSetPos:=arrAxisCtrl[VirAxisNo.P2M1_VirMain].Cmd.fSetPos;
//D_Sys.bP2M1Enable:=P2M1_MachCtrl.U.DT_ModelChees;

IF P2M1_MachCtrl.U.DT_iMode=1 THEN
	D_Sys.bP2M1Enable:=TRUE;	
ELSE
	D_Sys.bP2M1Enable:=FALSE;
END_IF

D_Sys.fM1MainSetPos:=arrAxis[P2M1_Axise.VirAxisName.VirMain].NcToPlc.SetPos;//1号叠片主虚轴位置 20240509 CF 
D_Pro.bAn_M1LockReady:=P2M1_MachCtrl.An_b.GetPiceReady;//正极取流水线极片准备好
D_Pro.bAn_M1JumpReady:=P2M1_MachCtrl.An_b.JumpPiceReady OR (bDiffVel[1] AND NOT P2M1_MachCtrl.An_b.GetPiceReady);//正极跳过取流水线极片准备好 20240509 CF
D_Pro.bCa_M1LockReady:=P2M1_MachCtrl.Ca_b.GetPiceReady;//负极取流水线极片准备好
D_Pro.bCa_M1JumpReady:=P2M1_MachCtrl.Ca_b.JumpPiceReady;//负极跳过取流水线极片准备好
D_Pro.bAn_M1PoleHave:=P2M1_MachCtrl.An_b.bAn_PoleHave;
D_Pro.bCa_M1PoleHave:=P2M1_MachCtrl.Ca_b.bCa_PoleHave;
//模切给叠片的信号
P2M1_MachCtrl.An_b.An_MainBeltOK:=M_Pro.bAn_M1Allow;//允许正极取极片
P2M1_MachCtrl.Ca_b.Ca_MainBeltOK:=M_Pro.bCa_M1Allow;//允许负极取极片
P2M1_MachCtrl.DTRunStatus.ReadyAllow2:=M_Pro.bAn_M1Allow2;

//运行时间统计
	DT1_Timedata(
							Alm:=P2M1_DTSysState.bErrorStop AND NOT P2M1_DError AND NOT P2M1_MachCtrl.DT_b.DT_GMchange (*OR  P2M1_WJSysState.bErrorStop*) , 
							Wait:= P2M1_MachCtrl.U.DT_iMode=3 AND NOT P2M1_MachCtrl.DT_b.DT_GMchange AND (NOT P2M1_DTSysState.bErrorStop OR P2M1_DError (* AND NOT  P2M1_WJSysState.bErrorStop*) )  , 
							Run:= P2M1_MachCtrl.U.DT_iMode=1 (*AND P2M1_MachCtrl.U.WJ_iMode=1 AND P2M1_MachCtrl.U.TJ_iMode=1*), 
							Overhang_NG:= P2M1_MachCtrl.DT_b.DT_OverhangNG, 
							GM_change:=P2M1_MachCtrl.DT_b.DT_GMchange, 
							Query:=P2M1_MachCtrl.DT_b.Query, 
							date1:=P2M1_MachCtrl.DT_b.date1 , 	
							STTimedata=> );

//屏蔽信号链接

//隔膜物料码OK
IF  (P3_PLC_PC_MES.Mes_PcToPlc5 AND  LEN(P3_PLC_PC_MES.Station1_Code)>6  ) OR P2M1_MachCtrl.DT_b.PartNumberOff THEN
	P2M1_MachCtrl.DT_b.DiaphragmPartNumberOK:=TRUE;
ELSE
	P2M1_MachCtrl.DT_b.DiaphragmPartNumberOK:=FALSE;
END_IF
//蓝胶物料码OK
IF  (P3_PLC_PC_MES.Mes_PcToPlc8 AND  LEN(P3_PLC_PC_MES.Station1_BlueCode)>6  ) OR P2M1_MachCtrl.DT_b.PartNumberOff THEN
	P2M1_MachCtrl.DT_b.BluePartNumberOK:=TRUE;
ELSE
	P2M1_MachCtrl.DT_b.BluePartNumberOK:=FALSE;
END_IF



IF P2M1_MachCtrl.DT_b.DiaphragmPartNumberOK THEN//隔膜料号OK
	CellMemory[P2M1_MachCtrl.DT_b.DT_Memory].Station_Code :=P3_PLC_PC_MES.Station1_Code;	
ELSE
	CellMemory[P2M1_MachCtrl.DT_b.DT_Memory].Station_Code :='';	
END_IF
IF P2M1_MachCtrl.DT_b.BluePartNumberOK THEN//蓝胶料号OK
	CellMemory[P2M1_MachCtrl.DT_b.DT_Memory].Station_BlueCode :=P3_PLC_PC_MES.Station1_BlueCode;	
ELSE
	CellMemory[P2M1_MachCtrl.DT_b.DT_Memory].Station_BlueCode :='';	
END_IF


	
//物料码清理
//隔膜条码重新校验
DT1Code_MES[1](CLK:=arrCyCtrl[P2M1_CycNo.CylinderName.PoleInflationCy].Status.ONState  , Q=> );  
IF DT1Code_MES[1].Q THEN
	P2M1_MachCtrl.DT_b.DiaphragmPartNumberOK:=FALSE;
	P3_PLC_PC_MES.Station1_Code:='';
	P3_PLC_PC_MES.Mes_PcToPlc5:=FALSE;
END_IF	

//蓝胶条码重新校验
DT1Code_MES[2](CLK:= P2M1_MachCtrl.DT_b.HMI_WinBtn[1] , Q=> );  
IF DT1Code_MES[2].Q THEN
	P2M1_MachCtrl.DT_b.BluePartNumberOK:=FALSE;
	P3_PLC_PC_MES.Station1_BlueCode:='';
	P3_PLC_PC_MES.Mes_PcToPlc8:=FALSE;
END_IF	

(*	
//物料码校验报警
IF NOT P2M1_MachCtrl.DT_b.DiaphragmPartNumberOK AND NOT P2M1_MachCtrl.DT_b.PartNumberOff THEN
	P2M1_MachCtrl.DT_b.Error[55]:=TRUE;//叠台隔膜物料码校验未通过，请重新校验物料码
END_IF
IF NOT P2M1_MachCtrl.DT_b.BluePartNumberOK AND NOT P2M1_MachCtrl.DT_b.PartNumberOff THEN
	P2M1_MachCtrl.DT_b.Error[56]:=TRUE;//叠台蓝胶物料码校验未通过，请重新校验物料码
END_IF

*)
	
	IF P2Btn.P2M1_Autobtn THEN
    arrCyCtrl[132].Cmd.bOFF:=TRUE;//1号叠台		隔膜接带平台除尘
    arrCyCtrl[132].Cmd.bON:=FALSE;
	ELSE
	   arrCyCtrl[132].Cmd.bON:=TRUE;
	   arrCyCtrl[132].Cmd.bOFF:=FALSE;
	END_IF

END_PROGRAM

// ---- P2POUs/POUS/P2M2_Auto.TcPOU
PROGRAM P2M2_Auto
VAR
	DT2Code_MES: ARRAY[1..10] OF R_TRIG;
END_VAR



// 2号叠台自动
P2M2_program(
	DTselect:=2, 
	Sys_Control:=P2M2_sysControl , 
	Mach_Control:=P2M2_MachCtrl , 
	arrCyNo:=P2M2_CycNo , 
	AxiseNo:=P2M2_Axise ,
	TableNo:=P2M2_TableNo, 
	Par:=P2M2_Par,CCD:=
	P2M2_CCD,
	Torque:=P2M2_Torque,
	iTargetTorqueTest=>iTargetTorque[2] );
	
//叠片给模切的信号
D_Pro.bAn_M2Done:=P2M2_MachCtrl.An_b.AN_BeltDone; //正极取流水线极片完成
D_Pro.bAn_M2Safety:=P2M2_MachCtrl.An_b.AN_BeltSafe;//正极取流水线安全位
D_Pro.bCa_M2Done:=P2M2_MachCtrl.Ca_b.Ca_BeltDone;//负极取水线极片完成
D_Pro.bCa_M2Safety:=P2M2_MachCtrl.Ca_b.Ca_BeltSafe;//负极取流水线安全位
//D_Sys.fM2MainSetPos:=arrAxisCtrl[VirAxisNo.P2M2_VirMain].Cmd.fSetPos;
//D_Sys.bP2M2Enable:=P2M2_MachCtrl.U.DT_ModelChees;

